       "CallManualOperationLines_ServoPos64Commands"(ManualOperationControl := "ManualOperationControl_U1Em5".axis64Pos[7].commands,
                                                     HmiInterface => "Unit1.Em5.HmiInterface".cmCathodeMainPnP2AxisX.commands);

       "CallManualOperationLines_ServoPos64Commands"(ManualOperationControl := "ManualOperationControl_U1Em5".axis64Pos[8].commands,
                                                     HmiInterface => "Unit1.Em5.HmiInterface".cmCathodeMainPnP1AxisY.commands);

       "CallManualOperationLines_ServoPos64Commands"(ManualOperationControl := "ManualOperationControl_U1Em5".axis64Pos[9].commands,
                                                     HmiInterface => "Unit1.Em5.HmiInterface".cmCathodeMainPnP1AxisZ.commands);

       "CallManualOperationLines_ServoPos64Commands"(ManualOperationControl := "ManualOperationControl_U1Em5".axis64Pos[10].commands,
                                                     HmiInterface => "Unit1.Em5.HmiInterface".cmCathodeMainPnP2AxisZ.commands);

       "CallManualOperationLines_ServoPos64Commands"(ManualOperationControl := "ManualOperationControl_U1Em5".axis64Pos[11].commands,
                                                     HmiInterface => "Unit1.Em5.HmiInterface".cmCathodeAlignTableAxisX.commands);

       "CallManualOperationLines_ServoPos64Commands"(ManualOperationControl := "ManualOperationControl_U1Em5".axis64Pos[12].commands,
                                                     HmiInterface => "Unit1.Em5.HmiInterface".cmCathodeAlignTableAxisY1.commands);

       "CallManualOperationLines_ServoPos64Commands"(ManualOperationControl := "ManualOperationControl_U1Em5".axis64Pos[13].commands,
                                                     HmiInterface => "Unit1.Em5.HmiInterface".cmCathodeAlignTableAxisY2.commands);

       // TwoWayActuator
       "Unit1.Em5.HmiInterface".cmCathodeMainPnP1RotaryCwCcw.commands := "ManualOperationControl_U1Em5".twoWayActuator[1].commands;
       "Unit1.Em5.HmiInterface".cmCathodeMainPnP1SuctionPlateVacuum.commands := "ManualOperationControl_U1Em5".twoWayActuator[2].commands;
       "Unit1.Em5.HmiInterface".cmCathodeMainPnP2SuctionPlateVacuum.commands := "ManualOperationControl_U1Em5".twoWayActuator[3].commands;
       "Unit1.Em5.HmiInterface".cmCathodeAlignTableSuctionPlateVacuum.commands := "ManualOperationControl_U1Em5".twoWayActuator[4].commands;
       "Unit1.Em5.HmiInterface".cmCathodeGlassCleaning.commands := "ManualOperationControl_U1Em5".twoWayActuator[5].commands;
       "Unit1.Em5.HmiInterface".cmCathodeNgPnpUpDown.commands := "ManualOperationControl_U1Em5".twoWayActuator[6].commands;
       "Unit1.Em5.HmiInterface".cmCathodeNgPnp1stFwdBwd.commands := "ManualOperationControl_U1Em5".twoWayActuator[7].commands;
       "Unit1.Em5.HmiInterface".cmCathodeNgPnp2ndFwdBwd.commands := "ManualOperationControl_U1Em5".twoWayActuator[8].commands;
       "Unit1.Em5.HmiInterface".cmCathodeMaintenanceMovingFixFrontRearFwdBwd.commands := "ManualOperationControl_U1Em5".twoWayActuator[9].commands;
       "Unit1.Em5.HmiInterface".cmCathodeNgBoxLiftUpDown.commands := "ManualOperationControl_U1Em5".twoWayActuator[10].commands;
       "Unit1.Em5.HmiInterface".cmCathodeNgBoxLockUpDown.commands := "ManualOperationControl_U1Em5".twoWayActuator[11].commands;
       "Unit1.Em5.HmiInterface".cmCathodeNgPnpVaccum.commands := "ManualOperationControl_U1Em5".twoWayActuator[12].commands;
       "Unit1.Em5.HmiInterface".cmCathodeConveyorCoverFwdBwd.commands := "ManualOperationControl_U1Em5".twoWayActuator[13].commands;

   END_REGION
END_REGION

REGION Network 13: Equipment Module 5
   RUNG wire#powerrail
      "CallManualOperationLines_EM"(disableUnit := #disableUnit1, manualOperationEm := "ManualOperationControl_U1Em5".manualOperationEm, manualOperationEmArea := "ManualOperationControl_U1Em5".manualOperationEmArea, manualOperationCms := "ManualOperationControl_U1Em5".manualOperationCms, Axis := "ManualOperationControl_U1Em5".axis, Axis64Pos := "ManualOperationControl_U1Em5".axis64Pos, AxisSfotCam := "ManualOperationControl_U1Em5".softCam, twoWayAcutor := "ManualOperationControl_U1Em5".twoWayActuator, Status := #StatusEm[5].Status, errorID := #errorIDEm[5].errorID)
   END_RUNG
   // the same network as SCL:
   "CallManualOperationLines_EM"(disableUnit := #disableUnit1,
                           manualOperationEm := "ManualOperationControl_U1Em5".manualOperationEm,
                           manualOperationEmArea := "ManualOperationControl_U1Em5".manualOperationEmArea,
                           manualOperationCms := "ManualOperationControl_U1Em5".manualOperationCms,
                           Axis := "ManualOperationControl_U1Em5".axis,
                           Axis64Pos := "ManualOperationControl_U1Em5".axis64Pos,
                           AxisSfotCam := "ManualOperationControl_U1Em5".softCam,
                           twoWayAcutor := "ManualOperationControl_U1Em5".twoWayActuator,
                           Status := #StatusEm[5].Status,
                           errorID := #errorIDEm[5].errorID);
END_REGION

REGION Network 14 (SCL): Equipment Module 6 Cms Mapping
   REGION Input Mapping
       // Axis
       "ManualOperationControl_U1Em6".axis64Pos[6].monitoring := "Unit1.Em6.HmiInterface".cmFinalRollerFrontAxisX.monitoring;
       "ManualOperationControl_U1Em6".axis64Pos[7].monitoring := "Unit1.Em6.HmiInterface".cmFinalRollerRearAxisX.monitoring;
       "ManualOperationControl_U1Em6".axis64Pos[8].monitoring := "Unit1.Em6.HmiInterface".cmMendrelCathodeFrontAxisY.monitoring;
       "ManualOperationControl_U1Em6".axis64Pos[9].monitoring := "Unit1.Em6.HmiInterface".cmMendrelCathodeFrontAxisZ.monitoring;
       "ManualOperationControl_U1Em6".axis64Pos[10].monitoring := "Unit1.Em6.HmiInterface".cmMendrelAnodeFrontAxisY.monitoring;
       "ManualOperationControl_U1Em6".axis64Pos[11].monitoring := "Unit1.Em6.HmiInterface".cmMendrelAnodeFrontAxisZ.monitoring;
       "ManualOperationControl_U1Em6".axis64Pos[12].monitoring := "Unit1.Em6.HmiInterface".cmMendrelCathodeRearAxisY.monitoring;
       "ManualOperationControl_U1Em6".axis64Pos[13].monitoring := "Unit1.Em6.HmiInterface".cmMendrelCathodeRearAxisZ.monitoring;
       "ManualOperationControl_U1Em6".axis64Pos[14].monitoring := "Unit1.Em6.HmiInterface".cmMendrelAnodeRearAxisY.monitoring;
       "ManualOperationControl_U1Em6".axis64Pos[15].monitoring := "Unit1.Em6.HmiInterface".cmMendrelAnodeRearAxisZ.monitoring;
       "ManualOperationControl_U1Em6".axis64Pos[16].monitoring := "Unit1.Em6.HmiInterface".cmStackTableAxisZ.monitoring;
       "ManualOperationControl_U1Em6".axis64Pos[17].monitoring := "Unit1.Em6.HmiInterface".cmStackTableOutFrontAxisZ.monitoring;
       "ManualOperationControl_U1Em6".axis64Pos[18].monitoring := "Unit1.Em6.HmiInterface".cmStackTableOutRearAxisZ.monitoring;

       "ManualOperationControl_U1Em6".axis64Pos[6].configuration := "Unit1.Em6.HmiInterface".cmFinalRollerFrontAxisX.configuration;
       "ManualOperationControl_U1Em6".axis64Pos[7].configuration := "Unit1.Em6.HmiInterface".cmFinalRollerRearAxisX.configuration;
       "ManualOperationControl_U1Em6".axis64Pos[8].configuration := "Unit1.Em6.HmiInterface".cmMendrelCathodeFrontAxisY.configuration;
       "ManualOperationControl_U1Em6".axis64Pos[9].configuration := "Unit1.Em6.HmiInterface".cmMendrelCathodeFrontAxisZ.configuration;
       "ManualOperationControl_U1Em6".axis64Pos[10].configuration := "Unit1.Em6.HmiInterface".cmMendrelAnodeFrontAxisY.configuration;
       "ManualOperationControl_U1Em6".axis64Pos[11].configuration := "Unit1.Em6.HmiInterface".cmMendrelAnodeFrontAxisZ.configuration;
       "ManualOperationControl_U1Em6".axis64Pos[12].configuration := "Unit1.Em6.HmiInterface".cmMendrelCathodeRearAxisY.configuration;
       "ManualOperationControl_U1Em6".axis64Pos[13].configuration := "Unit1.Em6.HmiInterface".cmMendrelCathodeRearAxisZ.configuration;
       "ManualOperationControl_U1Em6".axis64Pos[14].configuration := "Unit1.Em6.HmiInterface".cmMendrelAnodeRearAxisY.configuration;
       "ManualOperationControl_U1Em6".axis64Pos[15].configuration := "Unit1.Em6.HmiInterface".cmMendrelAnodeRearAxisZ.configuration;
       "ManualOperationControl_U1Em6".axis64Pos[16].configuration := "Unit1.Em6.HmiInterface".cmStackTableAxisZ.configuration;
       "ManualOperationControl_U1Em6".axis64Pos[17].configuration := "Unit1.Em6.HmiInterface".cmStackTableOutFrontAxisZ.configuration;
       "ManualOperationControl_U1Em6".axis64Pos[18].configuration := "Unit1.Em6.HmiInterface".cmStackTableOutRearAxisZ.configuration;

       // SoftCam
       "ManualOperationControl_U1Em6".softCam[6] := "Unit1.Em6.HmiInterface".cm.softCam.finalRollerFrontAxisX;
       "ManualOperationControl_U1Em6".softCam[7] := "Unit1.Em6.HmiInterface".cm.softCam.finalRollerRearAxisX;
       "ManualOperationControl_U1Em6".softCam[8] := "Unit1.Em6.HmiInterface".cm.softCam.mendrelAnodeFrontAxisY;
       "ManualOperationControl_U1Em6".softCam[9] := "Unit1.Em6.HmiInterface".cm.softCam.mendrelAnodeFrontAxisZ;
       "ManualOperationControl_U1Em6".softCam[10] := "Unit1.Em6.HmiInterface".cm.softCam.mendrelAnodeRearAxisY;
       "ManualOperationControl_U1Em6".softCam[11] := "Unit1.Em6.HmiInterface".cm.softCam.mendrelAnodeRearAxisZ;
       "ManualOperationControl_U1Em6".softCam[12] := "Unit1.Em6.HmiInterface".cm.softCam.mendrelCathodeFrontAxisY;
       "ManualOperationControl_U1Em6".softCam[13] := "Unit1.Em6.HmiInterface".cm.softCam.mendrelCathodeFrontAxisZ;
       "ManualOperationControl_U1Em6".softCam[14] := "Unit1.Em6.HmiInterface".cm.softCam.mendrelCathodeRearAxisY;
       "ManualOperationControl_U1Em6".softCam[15] := "Unit1.Em6.HmiInterface".cm.softCam.mendrelCathodeRearAxisZ;
       "ManualOperationControl_U1Em6".softCam[16] := "Unit1.Em6.HmiInterface".cm.softCam.stackTableAxisZ;
       "ManualOperationControl_U1Em6".softCam[17] := "Unit1.Em6.HmiInterface".cm.softCam.stackTableOutFrontAxisZ;
       "ManualOperationControl_U1Em6".softCam[18] := "Unit1.Em6.HmiInterface".cm.softCam.stackTableOutRearAxisZ;

       // TwoWayActuator
       "ManualOperationControl_U1Em6".twoWayActuator[1].monitoring := "Unit1.Em6.HmiInterface".cmMendrelCathodeFrontClamp.monitoring;
       "ManualOperationControl_U1Em6".twoWayActuator[2].monitoring := "Unit1.Em6.HmiInterface".cmMendrelAnodeFrontClamp.monitoring;
       "ManualOperationControl_U1Em6".twoWayActuator[3].monitoring := "Unit1.Em6.HmiInterface".cmMendrelCathodeRearClamp.monitoring;
       "ManualOperationControl_U1Em6".twoWayActuator[4].monitoring := "Unit1.Em6.HmiInterface".cmMendrelAnodeRearClamp.monitoring;
       "ManualOperationControl_U1Em6".twoWayActuator[5].monitoring := "Unit1.Em6.HmiInterface".cmStackTableVaccum.monitoring;
       "ManualOperationControl_U1Em6".twoWayActuator[6].monitoring := "Unit1.Em6.HmiInterface".cmStackTableGapPadUpDown.monitoring;

   END_REGION


   REGION Output Mapping
       // Axis
       "CallManualOperationLines_ServoPos64Commands"(ManualOperationControl := "ManualOperationControl_U1Em6".axis64Pos[6].commands,
                                                     HmiInterface => "Unit1.Em6.HmiInterface".cmFinalRollerFrontAxisX.commands);

       "CallManualOperationLines_ServoPos64Commands"(ManualOperationControl := "ManualOperationControl_U1Em6".axis64Pos[7].commands,
                                                     HmiInterface => "Unit1.Em6.HmiInterface".cmFinalRollerRearAxisX.commands);

       "CallManualOperationLines_ServoPos64Commands"(ManualOperationControl := "ManualOperationControl_U1Em6".axis64Pos[8].commands,
                                                     HmiInterface => "Unit1.Em6.HmiInterface".cmMendrelCathodeFrontAxisY.commands);

       "CallManualOperationLines_ServoPos64Commands"(ManualOperationControl := "ManualOperationControl_U1Em6".axis64Pos[9].commands,
                                                     HmiInterface => "Unit1.Em6.HmiInterface".cmMendrelCathodeFrontAxisZ.commands);

       "CallManualOperationLines_ServoPos64Commands"(ManualOperationControl := "ManualOperationControl_U1Em6".axis64Pos[10].commands,
                                                     HmiInterface => "Unit1.Em6.HmiInterface".cmMendrelAnodeFrontAxisY.commands);

       "CallManualOperationLines_ServoPos64Commands"(ManualOperationControl := "ManualOperationControl_U1Em6".axis64Pos[11].commands,
                                                     HmiInterface => "Unit1.Em6.HmiInterface".cmMendrelAnodeFrontAxisZ.commands);

       "CallManualOperationLines_ServoPos64Commands"(ManualOperationControl := "ManualOperationControl_U1Em6".axis64Pos[12].commands,
                                                     HmiInterface => "Unit1.Em6.HmiInterface".cmMendrelCathodeRearAxisY.commands);

       "CallManualOperationLines_ServoPos64Commands"(ManualOperationControl := "ManualOperationControl_U1Em6".axis64Pos[13].commands,
                                                     HmiInterface => "Unit1.Em6.HmiInterface".cmMendrelCathodeRearAxisZ.commands);

       "CallManualOperationLines_ServoPos64Commands"(ManualOperationControl := "ManualOperationControl_U1Em6".axis64Pos[14].commands,
                                                     HmiInterface => "Unit1.Em6.HmiInterface".cmMendrelAnodeRearAxisY.commands);

       "CallManualOperationLines_ServoPos64Commands"(ManualOperationControl := "ManualOperationControl_U1Em6".axis64Pos[15].commands,
                                                     HmiInterface => "Unit1.Em6.HmiInterface".cmMendrelAnodeRearAxisZ.commands);

       "CallManualOperationLines_ServoPos64Commands"(ManualOperationControl := "ManualOperationControl_U1Em6".axis64Pos[16].commands,
                                                     HmiInterface => "Unit1.Em6.HmiInterface".cmStackTableAxisZ.commands);

       "CallManualOperationLines_ServoPos64Commands"(ManualOperationControl := "ManualOperationControl_U1Em6".axis64Pos[17].commands,
                                                     HmiInterface => "Unit1.Em6.HmiInterface".cmStackTableOutFrontAxisZ.commands);

       "CallManualOperationLines_ServoPos64Commands"(ManualOperationControl := "ManualOperationControl_U1Em6".axis64Pos[18].commands,
                                                     HmiInterface => "Unit1.Em6.HmiInterface".cmStackTableOutRearAxisZ.commands);

       // TwoWayActuator
       "Unit1.Em6.HmiInterface".cmMendrelCathodeFrontClamp.commands := "ManualOperationControl_U1Em6".twoWayActuator[1].commands;
       "Unit1.Em6.HmiInterface".cmMendrelAnodeFrontClamp.commands := "ManualOperationControl_U1Em6".twoWayActuator[2].commands;
       "Unit1.Em6.HmiInterface".cmMendrelCathodeRearClamp.commands := "ManualOperationControl_U1Em6".twoWayActuator[3].commands;
       "Unit1.Em6.HmiInterface".cmMendrelAnodeRearClamp.commands := "ManualOperationControl_U1Em6".twoWayActuator[4].commands;
       "Unit1.Em6.HmiInterface".cmStackTableVaccum.commands := "ManualOperationControl_U1Em6".twoWayActuator[5].commands;
       "Unit1.Em6.HmiInterface".cmStackTableGapPadUpDown.commands := "ManualOperationControl_U1Em6".twoWayActuator[6].commands;
   END_REGION
END_REGION

REGION Network 15: Equipment Module 6
   RUNG wire#powerrail
      "CallManualOperationLines_EM"(disableUnit := #disableUnit1, manualOperationEm := "ManualOperationControl_U1Em6".manualOperationEm, manualOperationEmArea := "ManualOperationControl_U1Em6".manualOperationEmArea, manualOperationCms := "ManualOperationControl_U1Em6".manualOperationCms, Axis := "ManualOperationControl_U1Em6".axis, Axis64Pos := "ManualOperationControl_U1Em6".axis64Pos, AxisSfotCam := "ManualOperationControl_U1Em6".softCam, twoWayAcutor := "ManualOperationControl_U1Em6".twoWayActuator, Status := #StatusEm[6].Status, errorID := #errorIDEm[6].errorID)
   END_RUNG
   // the same network as SCL:
   "CallManualOperationLines_EM"(disableUnit := #disableUnit1,
                           manualOperationEm := "ManualOperationControl_U1Em6".manualOperationEm,
                           manualOperationEmArea := "ManualOperationControl_U1Em6".manualOperationEmArea,
                           manualOperationCms := "ManualOperationControl_U1Em6".manualOperationCms,
                           Axis := "ManualOperationControl_U1Em6".axis,
                           Axis64Pos := "ManualOperationControl_U1Em6".axis64Pos,
                           AxisSfotCam := "ManualOperationControl_U1Em6".softCam,
                           twoWayAcutor := "ManualOperationControl_U1Em6".twoWayActuator,
                           Status := #StatusEm[6].Status,
                           errorID := #errorIDEm[6].errorID);
END_REGION

REGION Network 16 (SCL): Equipment Module 7 Cms Mapping
   REGION Input Mapping
       // Axis
       "ManualOperationControl_U1Em7".axis64Pos[6].monitoring := "Unit1.Em7.HmiInterface".cmSepaClampnCutterAxisX.monitoring;
       "ManualOperationControl_U1Em7".axis64Pos[7].monitoring := "Unit1.Em7.HmiInterface".cmSepaClampnCutterAxisZ.monitoring;
       "ManualOperationControl_U1Em7".axis64Pos[8].monitoring := "Unit1.Em7.HmiInterface".cmSepaGripperAxisX.monitoring;
       "ManualOperationControl_U1Em7".axis64Pos[9].monitoring := "Unit1.Em7.HmiInterface".cmSepaGripperAxisZ.monitoring;
       "ManualOperationControl_U1Em7".axis64Pos[10].monitoring := "Unit1.Em7.HmiInterface".cmSepaGripperAxisC.monitoring;
       "ManualOperationControl_U1Em7".axis64Pos[11].monitoring := "Unit1.Em7.HmiInterface".cmJRWinderFrontAxisY.monitoring;
       "ManualOperationControl_U1Em7".axis64Pos[12].monitoring := "Unit1.Em7.HmiInterface".cmJRWinderRearAxisY.monitoring;
       "ManualOperationControl_U1Em7".axis64Pos[13].monitoring := "Unit1.Em7.HmiInterface".cmJRWinderAxisB.monitoring;
       "ManualOperationControl_U1Em7".axis64Pos[14].monitoring := "Unit1.Em7.HmiInterface".cmJRPusherAxisZ.monitoring;

       "ManualOperationControl_U1Em7".axis64Pos[6].configuration := "Unit1.Em7.HmiInterface".cmSepaClampnCutterAxisX.configuration;
       "ManualOperationControl_U1Em7".axis64Pos[7].configuration := "Unit1.Em7.HmiInterface".cmSepaClampnCutterAxisZ.configuration;
       "ManualOperationControl_U1Em7".axis64Pos[8].configuration := "Unit1.Em7.HmiInterface".cmSepaGripperAxisX.configuration;
       "ManualOperationControl_U1Em7".axis64Pos[9].configuration := "Unit1.Em7.HmiInterface".cmSepaGripperAxisZ.configuration;
       "ManualOperationControl_U1Em7".axis64Pos[10].configuration := "Unit1.Em7.HmiInterface".cmSepaGripperAxisC.configuration;
       "ManualOperationControl_U1Em7".axis64Pos[11].configuration := "Unit1.Em7.HmiInterface".cmJRWinderFrontAxisY.configuration;
       "ManualOperationControl_U1Em7".axis64Pos[12].configuration := "Unit1.Em7.HmiInterface".cmJRWinderRearAxisY.configuration;
       "ManualOperationControl_U1Em7".axis64Pos[13].configuration := "Unit1.Em7.HmiInterface".cmJRWinderAxisB.configuration;
       "ManualOperationControl_U1Em7".axis64Pos[14].configuration := "Unit1.Em7.HmiInterface".cmJRPusherAxisZ.configuration;

       // SoftCam
       "ManualOperationControl_U1Em7".softCam[6] := "Unit1.Em7.HmiInterface".cm.softCam.sepaClampnCutterAxisX;
       "ManualOperationControl_U1Em7".softCam[7] := "Unit1.Em7.HmiInterface".cm.softCam.sepaClampnCutterAxisZ;
       "ManualOperationControl_U1Em7".softCam[8] := "Unit1.Em7.HmiInterface".cm.softCam.sepaGripperAxisX;
       "ManualOperationControl_U1Em7".softCam[9] := "Unit1.Em7.HmiInterface".cm.softCam.sepaGripperAxisZ;
       "ManualOperationControl_U1Em7".softCam[10] := "Unit1.Em7.HmiInterface".cm.softCam.sepaGripperAxisC;
       "ManualOperationControl_U1Em7".softCam[11] := "Unit1.Em7.HmiInterface".cm.softCam.jrWinderRearAxisY;
       "ManualOperationControl_U1Em7".softCam[12] := "Unit1.Em7.HmiInterface".cm.softCam.jrWinderFrontAxisY;
       "ManualOperationControl_U1Em7".softCam[13] := "Unit1.Em7.HmiInterface".cm.softCam.jrWinderAxisB;
       "ManualOperationControl_U1Em7".softCam[14] := "Unit1.Em7.HmiInterface".cm.softCam.jrPusherAxisZ;

       // TwoWayActuator
       "ManualOperationControl_U1Em7".twoWayActuator[1].monitoring := "Unit1.Em7.HmiInterface".cmSepaCutterUpDown.monitoring;
       "ManualOperationControl_U1Em7".twoWayActuator[2].monitoring := "Unit1.Em7.HmiInterface".cmSepaClampTopUpDown.monitoring;
       "ManualOperationControl_U1Em7".twoWayActuator[3].monitoring := "Unit1.Em7.HmiInterface".cmSepaClampBottomUpDown.monitoring;
       "ManualOperationControl_U1Em7".twoWayActuator[4].monitoring := "Unit1.Em7.HmiInterface".cmStackGripperOpenClose.monitoring;
       "ManualOperationControl_U1Em7".twoWayActuator[5].monitoring := "Unit1.Em7.HmiInterface".cmStackGripperFwdBwd.monitoring;
       "ManualOperationControl_U1Em7".twoWayActuator[6].monitoring := "Unit1.Em7.HmiInterface".cmJRWinderClampTopRearUpDown.monitoring;
       "ManualOperationControl_U1Em7".twoWayActuator[7].monitoring := "Unit1.Em7.HmiInterface".cmJRWinderClampBtmRearUpDown.monitoring;
       "ManualOperationControl_U1Em7".twoWayActuator[8].monitoring := "Unit1.Em7.HmiInterface".cmJRWinderClampTopFrontUpDown.monitoring;
       "ManualOperationControl_U1Em7".twoWayActuator[9].monitoring := "Unit1.Em7.HmiInterface".cmJRWinderClampBtmFrontUpDown.monitoring;
       "ManualOperationControl_U1Em7".twoWayActuator[10].monitoring := "Unit1.Em7.HmiInterface".cmPusherRollerFwdBwd.monitoring;

   END_REGION


   REGION Output Mapping
       // Axis
       "CallManualOperationLines_ServoPos64Commands"(ManualOperationControl := "ManualOperationControl_U1Em7".axis64Pos[6].commands,
                                                     HmiInterface => "Unit1.Em7.HmiInterface".cmSepaClampnCutterAxisX.commands);

       "CallManualOperationLines_ServoPos64Commands"(ManualOperationControl := "ManualOperationControl_U1Em7".axis64Pos[7].commands,
                                                     HmiInterface => "Unit1.Em7.HmiInterface".cmSepaClampnCutterAxisZ.commands);

       "CallManualOperationLines_ServoPos64Commands"(ManualOperationControl := "ManualOperationControl_U1Em7".axis64Pos[8].commands,
                                                     HmiInterface => "Unit1.Em7.HmiInterface".cmSepaGripperAxisX.commands);

       "CallManualOperationLines_ServoPos64Commands"(ManualOperationControl := "ManualOperationControl_U1Em7".axis64Pos[9].commands,
                                                     HmiInterface => "Unit1.Em7.HmiInterface".cmSepaGripperAxisZ.commands);

       "CallManualOperationLines_ServoPos64Commands"(ManualOperationControl := "ManualOperationControl_U1Em7".axis64Pos[10].commands,
                                                     HmiInterface => "Unit1.Em7.HmiInterface".cmSepaGripperAxisC.commands);

       "CallManualOperationLines_ServoPos64Commands"(ManualOperationControl := "ManualOperationControl_U1Em7".axis64Pos[11].commands,
                                                     HmiInterface => "Unit1.Em7.HmiInterface".cmJRWinderFrontAxisY.commands);

       "CallManualOperationLines_ServoPos64Commands"(ManualOperationControl := "ManualOperationControl_U1Em7".axis64Pos[12].commands,
                                                     HmiInterface => "Unit1.Em7.HmiInterface".cmJRWinderRearAxisY.commands);

       "CallManualOperationLines_ServoPos64Commands"(ManualOperationControl := "ManualOperationControl_U1Em7".axis64Pos[13].commands,
                                                     HmiInterface => "Unit1.Em7.HmiInterface".cmJRWinderAxisB.commands);

       "CallManualOperationLines_ServoPos64Commands"(ManualOperationControl := "ManualOperationControl_U1Em7".axis64Pos[14].commands,
                                                     HmiInterface => "Unit1.Em7.HmiInterface".cmJRPusherAxisZ.commands);

       // TwoWayActuator
       "Unit1.Em7.HmiInterface".cmSepaCutterUpDown.commands := "ManualOperationControl_U1Em7".twoWayActuator[1].commands;
       "Unit1.Em7.HmiInterface".cmSepaClampTopUpDown.commands := "ManualOperationControl_U1Em7".twoWayActuator[2].commands;
       "Unit1.Em7.HmiInterface".cmSepaClampBottomUpDown.commands := "ManualOperationControl_U1Em7".twoWayActuator[3].commands;
       "Unit1.Em7.HmiInterface".cmStackGripperOpenClose.commands := "ManualOperationControl_U1Em7".twoWayActuator[4].commands;
       "Unit1.Em7.HmiInterface".cmStackGripperFwdBwd.commands := "ManualOperationControl_U1Em7".twoWayActuator[5].commands;
       "Unit1.Em7.HmiInterface".cmJRWinderClampTopRearUpDown.commands := "ManualOperationControl_U1Em7".twoWayActuator[6].commands;
       "Unit1.Em7.HmiInterface".cmJRWinderClampBtmRearUpDown.commands := "ManualOperationControl_U1Em7".twoWayActuator[7].commands;
       "Unit1.Em7.HmiInterface".cmJRWinderClampTopFrontUpDown.commands := "ManualOperationControl_U1Em7".twoWayActuator[8].commands;
       "Unit1.Em7.HmiInterface".cmJRWinderClampBtmFrontUpDown.commands := "ManualOperationControl_U1Em7".twoWayActuator[9].commands;
       "Unit1.Em7.HmiInterface".cmPusherRollerFwdBwd.commands := "ManualOperationControl_U1Em7".twoWayActuator[10].commands;

   END_REGION
END_REGION

REGION Network 17: Equipment Module 7
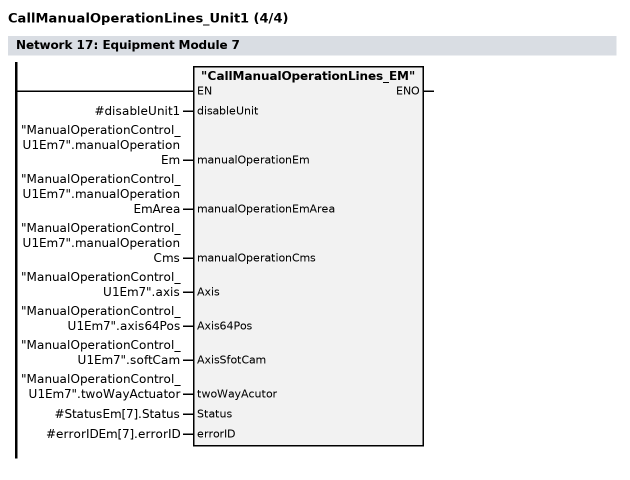
   RUNG wire#powerrail
      "CallManualOperationLines_EM"(disableUnit := #disableUnit1, manualOperationEm := "ManualOperationControl_U1Em7".manualOperationEm, manualOperationEmArea := "ManualOperationControl_U1Em7".manualOperationEmArea, manualOperationCms := "ManualOperationControl_U1Em7".manualOperationCms, Axis := "ManualOperationControl_U1Em7".axis, Axis64Pos := "ManualOperationControl_U1Em7".axis64Pos, AxisSfotCam := "ManualOperationControl_U1Em7".softCam, twoWayAcutor := "ManualOperationControl_U1Em7".twoWayActuator, Status := #StatusEm[7].Status, errorID := #errorIDEm[7].errorID)
   END_RUNG
   // the same network as SCL:
   "CallManualOperationLines_EM"(disableUnit := #disableUnit1,
                           manualOperationEm := "ManualOperationControl_U1Em7".manualOperationEm,
                           manualOperationEmArea := "ManualOperationControl_U1Em7".manualOperationEmArea,
                           manualOperationCms := "ManualOperationControl_U1Em7".manualOperationCms,
                           Axis := "ManualOperationControl_U1Em7".axis,
                           Axis64Pos := "ManualOperationControl_U1Em7".axis64Pos,
                           AxisSfotCam := "ManualOperationControl_U1Em7".softCam,
                           twoWayAcutor := "ManualOperationControl_U1Em7".twoWayActuator,
                           Status := #StatusEm[7].Status,
                           errorID := #errorIDEm[7].errorID);
END_REGION
END_FUNCTION

FUNCTION "CallManualOperationLines_EM" : Void   // FC82, LAD
// stored: SetENOAutomatically false
   VAR_INPUT
      disableUnit : Bool;
   END_VAR
   VAR_IN_OUT
      manualOperationEm : "LAF_typeManEm";
      manualOperationEmArea : Array[*] of "LAF_typeManOperationArea";
      manualOperationCms : Array[*] of "LAF_typeManOperation";
      Axis : Array[*] of "LBC_typeAxisControlInterface";
      Axis64Pos : Array[*] of "LBC_typeAxis64PosInterface";
      AxisSfotCam : Array[*] of "LER_typeSoftCamInterface2";
      twoWayAcutor : Array[*] of "LBC_typeTwoWayActuatorInterface";
      Status : Array[*] of Word;
      errorID : Array[*] of Word;
   END_VAR
   VAR_TEMP
      tempLowerBoundAxis : Int;
      tempUpperBoundAxis : Int;
      tempLowerBoundAxis64Pos : Int;
      tempUpperBoundAxis64Pos : Int;
      tempLowerBoundTwoWayAct : Int;
      tempUpperBoundTwoWayAct : Int;
      tempEnd : Bool;
   END_VAR
BEGIN

REGION Network 1: Detect lower and upper bound of the array for further processing
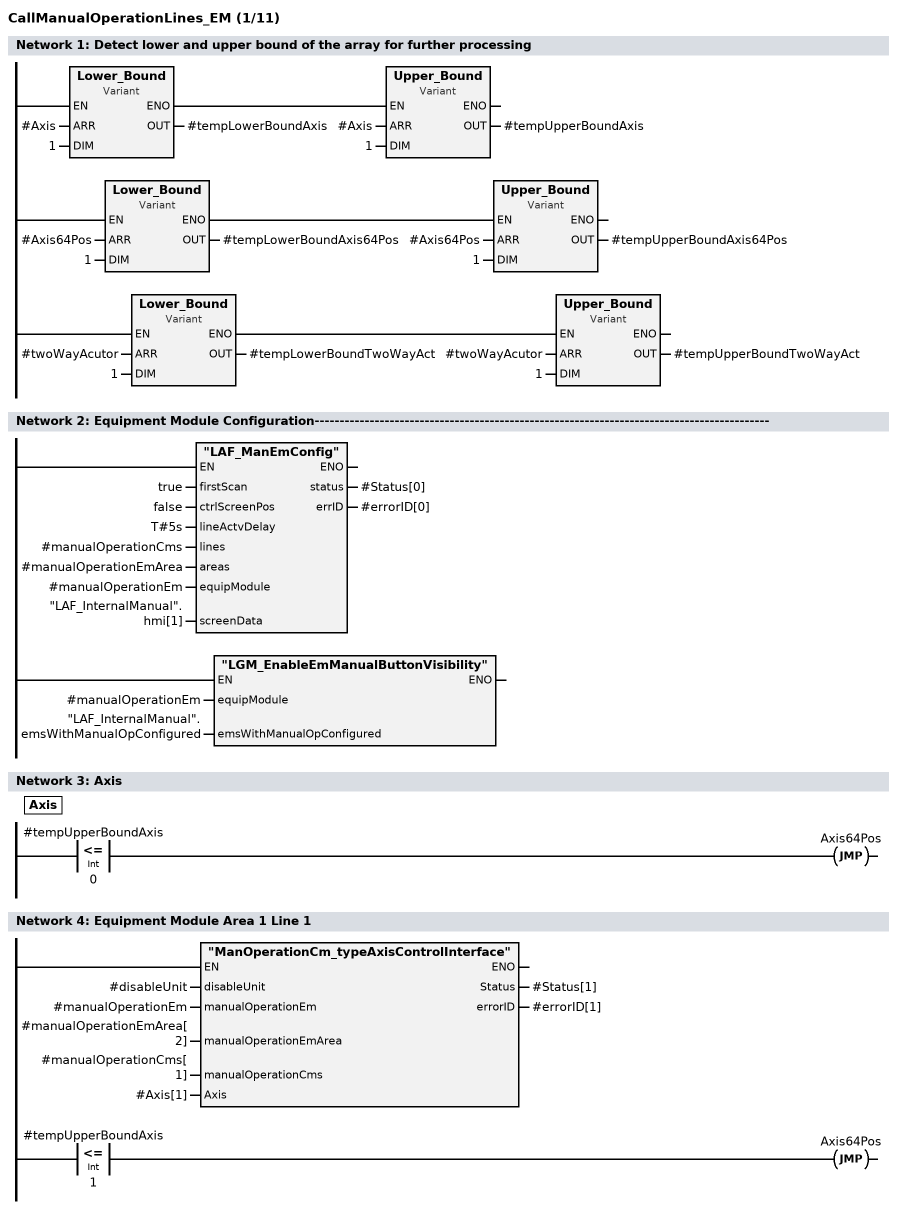
   // no SCL statement known for Lower_Bound, Upper_Bound: written as a call
   // ENO of a box is taken as its EN; it also drops when the box reports an error
   Lower_Bound(arr := #Axis, dim := 1, out => #tempLowerBoundAxis);
   Upper_Bound(arr := #Axis, dim := 1, out => #tempUpperBoundAxis);
   Lower_Bound(arr := #Axis64Pos, dim := 1, out => #tempLowerBoundAxis64Pos);
   Upper_Bound(arr := #Axis64Pos, dim := 1, out => #tempUpperBoundAxis64Pos);
   Lower_Bound(arr := #twoWayAcutor, dim := 1, out => #tempLowerBoundTwoWayAct);
   Upper_Bound(arr := #twoWayAcutor, dim := 1, out => #tempUpperBoundTwoWayAct);
END_REGION

REGION Network 2: Equipment Module Configuration-------------------------------------------------------------------------------------------
   RUNG wire#powerrail
      "LAF_ManEmConfig"(firstScan := true, ctrlScreenPos := false, lineActvDelay := T#5s, lines := #manualOperationCms, areas := #manualOperationEmArea, equipModule := #manualOperationEm, screenData := "LAF_InternalManual".hmi[1], status => #Status[0], errID => #errorID[0])
   END_RUNG
   RUNG wire#powerrail
      "LGM_EnableEmManualButtonVisibility"(equipModule := #manualOperationEm, emsWithManualOpConfigured := "LAF_InternalManual".emsWithManualOpConfigured)
   END_RUNG
   // the same network as SCL:
   "LAF_ManEmConfig"(firstScan := true,
                     ctrlScreenPos := false,
                     lineActvDelay := T#5s,
                     lines := #manualOperationCms,
                     areas := #manualOperationEmArea,
                     equipModule := #manualOperationEm,
                     screenData := "LAF_InternalManual".hmi[1],
                     status => #Status[0],
                     errID => #errorID[0]);
   "LGM_EnableEmManualButtonVisibility"(equipModule := #manualOperationEm,
                           emsWithManualOpConfigured := "LAF_InternalManual".emsWithManualOpConfigured);
END_REGION

REGION Network 3: Axis
   Label( Axis )
   RUNG wire#powerrail
      { S7_Templates := "SrcType := Int" } LE_Contact(in1 := #tempUpperBoundAxis, in2 := 0)
      JumpCoil( Axis64Pos )
   END_RUNG
   // the same network as SCL:
   Axis:
   IF #tempUpperBoundAxis <= 0 THEN GOTO Axis64Pos; END_IF;
END_REGION

REGION Network 4: Equipment Module Area 1 Line 1
   RUNG wire#powerrail
      "ManOperationCm_typeAxisControlInterface"(disableUnit := #disableUnit, manualOperationEm := #manualOperationEm, manualOperationEmArea := #manualOperationEmArea[2], manualOperationCms := #manualOperationCms[1], Axis := #Axis[1], Status => #Status[1], errorID => #errorID[1])
   END_RUNG
   RUNG wire#powerrail
      { S7_Templates := "SrcType := Int" } LE_Contact(in1 := #tempUpperBoundAxis, in2 := 1)
      JumpCoil( Axis64Pos )
   END_RUNG
   // the same network as SCL:
   "ManOperationCm_typeAxisControlInterface"(disableUnit := #disableUnit,
                           manualOperationEm := #manualOperationEm,
                           manualOperationEmArea := #manualOperationEmArea[2],
                           manualOperationCms := #manualOperationCms[1],
                           Axis := #Axis[1],
                           Status => #Status[1],
                           errorID => #errorID[1]);
   IF #tempUpperBoundAxis <= 1 THEN GOTO Axis64Pos; END_IF;
END_REGION

REGION Network 5: Equipment Module Area 1 Line 2
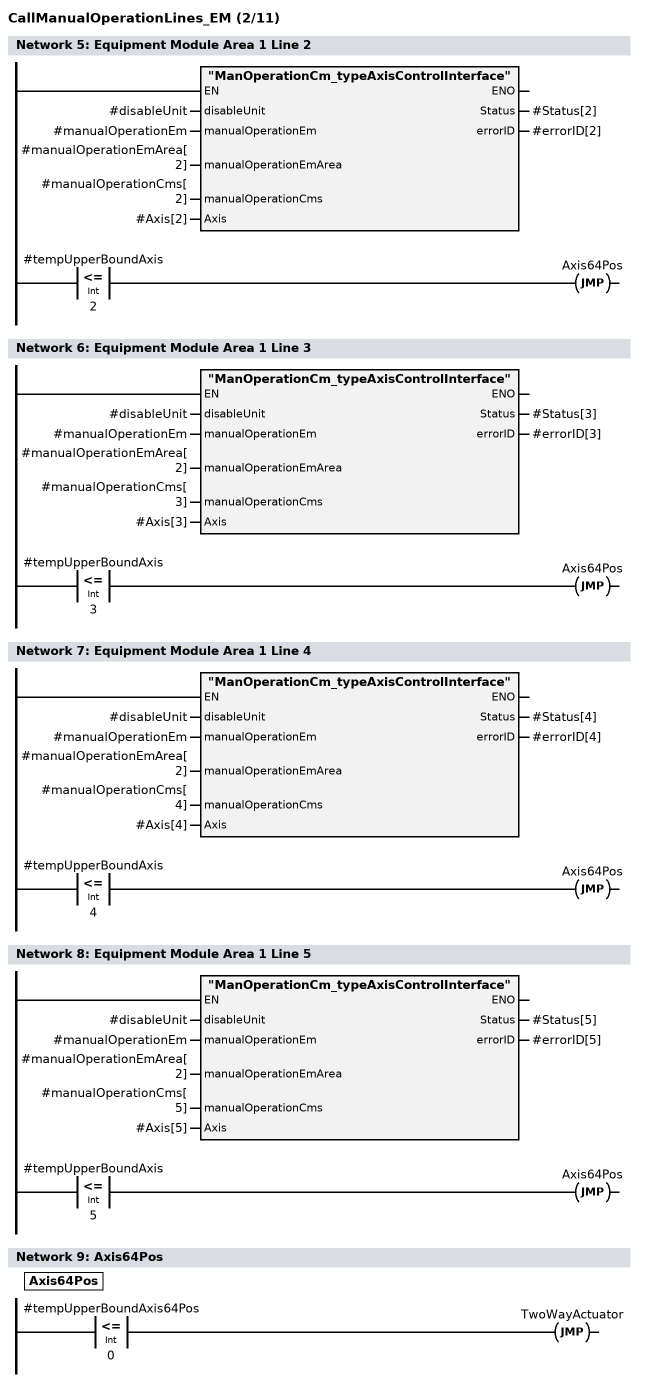
   RUNG wire#powerrail
      "ManOperationCm_typeAxisControlInterface"(disableUnit := #disableUnit, manualOperationEm := #manualOperationEm, manualOperationEmArea := #manualOperationEmArea[2], manualOperationCms := #manualOperationCms[2], Axis := #Axis[2], Status => #Status[2], errorID => #errorID[2])
   END_RUNG
   RUNG wire#powerrail
      { S7_Templates := "SrcType := Int" } LE_Contact(in1 := #tempUpperBoundAxis, in2 := 2)
      JumpCoil( Axis64Pos )
   END_RUNG
   // the same network as SCL:
   "ManOperationCm_typeAxisControlInterface"(disableUnit := #disableUnit,
                           manualOperationEm := #manualOperationEm,
                           manualOperationEmArea := #manualOperationEmArea[2],
                           manualOperationCms := #manualOperationCms[2],
                           Axis := #Axis[2],
                           Status => #Status[2],
                           errorID => #errorID[2]);
   IF #tempUpperBoundAxis <= 2 THEN GOTO Axis64Pos; END_IF;
END_REGION

REGION Network 6: Equipment Module Area 1 Line 3
   RUNG wire#powerrail
      "ManOperationCm_typeAxisControlInterface"(disableUnit := #disableUnit, manualOperationEm := #manualOperationEm, manualOperationEmArea := #manualOperationEmArea[2], manualOperationCms := #manualOperationCms[3], Axis := #Axis[3], Status => #Status[3], errorID => #errorID[3])
   END_RUNG
   RUNG wire#powerrail
      { S7_Templates := "SrcType := Int" } LE_Contact(in1 := #tempUpperBoundAxis, in2 := 3)
      JumpCoil( Axis64Pos )
   END_RUNG
   // the same network as SCL:
   "ManOperationCm_typeAxisControlInterface"(disableUnit := #disableUnit,
                           manualOperationEm := #manualOperationEm,
                           manualOperationEmArea := #manualOperationEmArea[2],
                           manualOperationCms := #manualOperationCms[3],
                           Axis := #Axis[3],
                           Status => #Status[3],
                           errorID => #errorID[3]);
   IF #tempUpperBoundAxis <= 3 THEN GOTO Axis64Pos; END_IF;
END_REGION

REGION Network 7: Equipment Module Area 1 Line 4
   RUNG wire#powerrail
      "ManOperationCm_typeAxisControlInterface"(disableUnit := #disableUnit, manualOperationEm := #manualOperationEm, manualOperationEmArea := #manualOperationEmArea[2], manualOperationCms := #manualOperationCms[4], Axis := #Axis[4], Status => #Status[4], errorID => #errorID[4])
   END_RUNG
   RUNG wire#powerrail
      { S7_Templates := "SrcType := Int" } LE_Contact(in1 := #tempUpperBoundAxis, in2 := 4)
      JumpCoil( Axis64Pos )
   END_RUNG
   // the same network as SCL:
   "ManOperationCm_typeAxisControlInterface"(disableUnit := #disableUnit,
                           manualOperationEm := #manualOperationEm,
                           manualOperationEmArea := #manualOperationEmArea[2],
                           manualOperationCms := #manualOperationCms[4],
                           Axis := #Axis[4],
                           Status => #Status[4],
                           errorID => #errorID[4]);
   IF #tempUpperBoundAxis <= 4 THEN GOTO Axis64Pos; END_IF;
END_REGION

REGION Network 8: Equipment Module Area 1 Line 5
   RUNG wire#powerrail
      "ManOperationCm_typeAxisControlInterface"(disableUnit := #disableUnit, manualOperationEm := #manualOperationEm, manualOperationEmArea := #manualOperationEmArea[2], manualOperationCms := #manualOperationCms[5], Axis := #Axis[5], Status => #Status[5], errorID => #errorID[5])
   END_RUNG
   RUNG wire#powerrail
      { S7_Templates := "SrcType := Int" } LE_Contact(in1 := #tempUpperBoundAxis, in2 := 5)
      JumpCoil( Axis64Pos )
   END_RUNG
   // the same network as SCL:
   "ManOperationCm_typeAxisControlInterface"(disableUnit := #disableUnit,
                           manualOperationEm := #manualOperationEm,
                           manualOperationEmArea := #manualOperationEmArea[2],
                           manualOperationCms := #manualOperationCms[5],
                           Axis := #Axis[5],
                           Status => #Status[5],
                           errorID => #errorID[5]);
   IF #tempUpperBoundAxis <= 5 THEN GOTO Axis64Pos; END_IF;
END_REGION

REGION Network 9: Axis64Pos
   Label( Axis64Pos )
   RUNG wire#powerrail
      { S7_Templates := "SrcType := Int" } LE_Contact(in1 := #tempUpperBoundAxis64Pos, in2 := 0)
      JumpCoil( TwoWayActuator )
   END_RUNG
   // the same network as SCL:
   Axis64Pos:
   IF #tempUpperBoundAxis64Pos <= 0 THEN GOTO TwoWayActuator; END_IF;
END_REGION

REGION Network 10: Equipment Module Area 1 Line 6
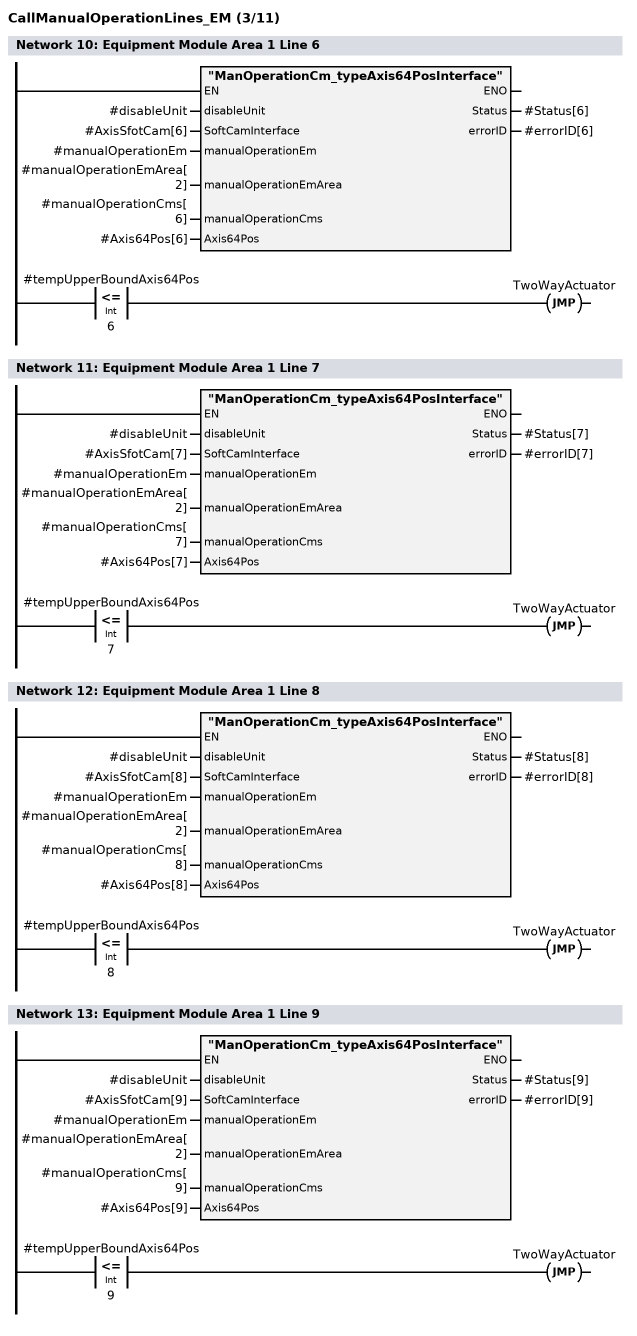
   RUNG wire#powerrail
      "ManOperationCm_typeAxis64PosInterface"(disableUnit := #disableUnit, SoftCamInterface := #AxisSfotCam[6], manualOperationEm := #manualOperationEm, manualOperationEmArea := #manualOperationEmArea[2], manualOperationCms := #manualOperationCms[6], Axis64Pos := #Axis64Pos[6], Status => #Status[6], errorID => #errorID[6])
   END_RUNG
   RUNG wire#powerrail
      { S7_Templates := "SrcType := Int" } LE_Contact(in1 := #tempUpperBoundAxis64Pos, in2 := 6)
      JumpCoil( TwoWayActuator )
   END_RUNG
   // the same network as SCL:
   "ManOperationCm_typeAxis64PosInterface"(disableUnit := #disableUnit,
                           SoftCamInterface := #AxisSfotCam[6],
                           manualOperationEm := #manualOperationEm,
                           manualOperationEmArea := #manualOperationEmArea[2],
                           manualOperationCms := #manualOperationCms[6],
                           Axis64Pos := #Axis64Pos[6],
                           Status => #Status[6],
                           errorID => #errorID[6]);
   IF #tempUpperBoundAxis64Pos <= 6 THEN GOTO TwoWayActuator; END_IF;
END_REGION

REGION Network 11: Equipment Module Area 1 Line 7
   RUNG wire#powerrail
      "ManOperationCm_typeAxis64PosInterface"(disableUnit := #disableUnit, SoftCamInterface := #AxisSfotCam[7], manualOperationEm := #manualOperationEm, manualOperationEmArea := #manualOperationEmArea[2], manualOperationCms := #manualOperationCms[7], Axis64Pos := #Axis64Pos[7], Status => #Status[7], errorID => #errorID[7])
   END_RUNG
   RUNG wire#powerrail
      { S7_Templates := "SrcType := Int" } LE_Contact(in1 := #tempUpperBoundAxis64Pos, in2 := 7)
      JumpCoil( TwoWayActuator )
   END_RUNG
   // the same network as SCL:
   "ManOperationCm_typeAxis64PosInterface"(disableUnit := #disableUnit,
                           SoftCamInterface := #AxisSfotCam[7],
                           manualOperationEm := #manualOperationEm,
                           manualOperationEmArea := #manualOperationEmArea[2],
                           manualOperationCms := #manualOperationCms[7],
                           Axis64Pos := #Axis64Pos[7],
                           Status => #Status[7],
                           errorID => #errorID[7]);
   IF #tempUpperBoundAxis64Pos <= 7 THEN GOTO TwoWayActuator; END_IF;
END_REGION

REGION Network 12: Equipment Module Area 1 Line 8
   RUNG wire#powerrail
      "ManOperationCm_typeAxis64PosInterface"(disableUnit := #disableUnit, SoftCamInterface := #AxisSfotCam[8], manualOperationEm := #manualOperationEm, manualOperationEmArea := #manualOperationEmArea[2], manualOperationCms := #manualOperationCms[8], Axis64Pos := #Axis64Pos[8], Status => #Status[8], errorID => #errorID[8])
   END_RUNG
   RUNG wire#powerrail
      { S7_Templates := "SrcType := Int" } LE_Contact(in1 := #tempUpperBoundAxis64Pos, in2 := 8)
      JumpCoil( TwoWayActuator )
   END_RUNG
   // the same network as SCL:
   "ManOperationCm_typeAxis64PosInterface"(disableUnit := #disableUnit,
                           SoftCamInterface := #AxisSfotCam[8],
                           manualOperationEm := #manualOperationEm,
                           manualOperationEmArea := #manualOperationEmArea[2],
                           manualOperationCms := #manualOperationCms[8],
                           Axis64Pos := #Axis64Pos[8],
                           Status => #Status[8],
                           errorID => #errorID[8]);
   IF #tempUpperBoundAxis64Pos <= 8 THEN GOTO TwoWayActuator; END_IF;
END_REGION

REGION Network 13: Equipment Module Area 1 Line 9
   RUNG wire#powerrail
      "ManOperationCm_typeAxis64PosInterface"(disableUnit := #disableUnit, SoftCamInterface := #AxisSfotCam[9], manualOperationEm := #manualOperationEm, manualOperationEmArea := #manualOperationEmArea[2], manualOperationCms := #manualOperationCms[9], Axis64Pos := #Axis64Pos[9], Status => #Status[9], errorID => #errorID[9])
   END_RUNG
   RUNG wire#powerrail
      { S7_Templates := "SrcType := Int" } LE_Contact(in1 := #tempUpperBoundAxis64Pos, in2 := 9)
      JumpCoil( TwoWayActuator )
   END_RUNG
   // the same network as SCL:
   "ManOperationCm_typeAxis64PosInterface"(disableUnit := #disableUnit,
                           SoftCamInterface := #AxisSfotCam[9],
                           manualOperationEm := #manualOperationEm,
                           manualOperationEmArea := #manualOperationEmArea[2],
                           manualOperationCms := #manualOperationCms[9],
                           Axis64Pos := #Axis64Pos[9],
                           Status => #Status[9],
                           errorID => #errorID[9]);
   IF #tempUpperBoundAxis64Pos <= 9 THEN GOTO TwoWayActuator; END_IF;
END_REGION

REGION Network 14: Equipment Module Area 1 Line 10
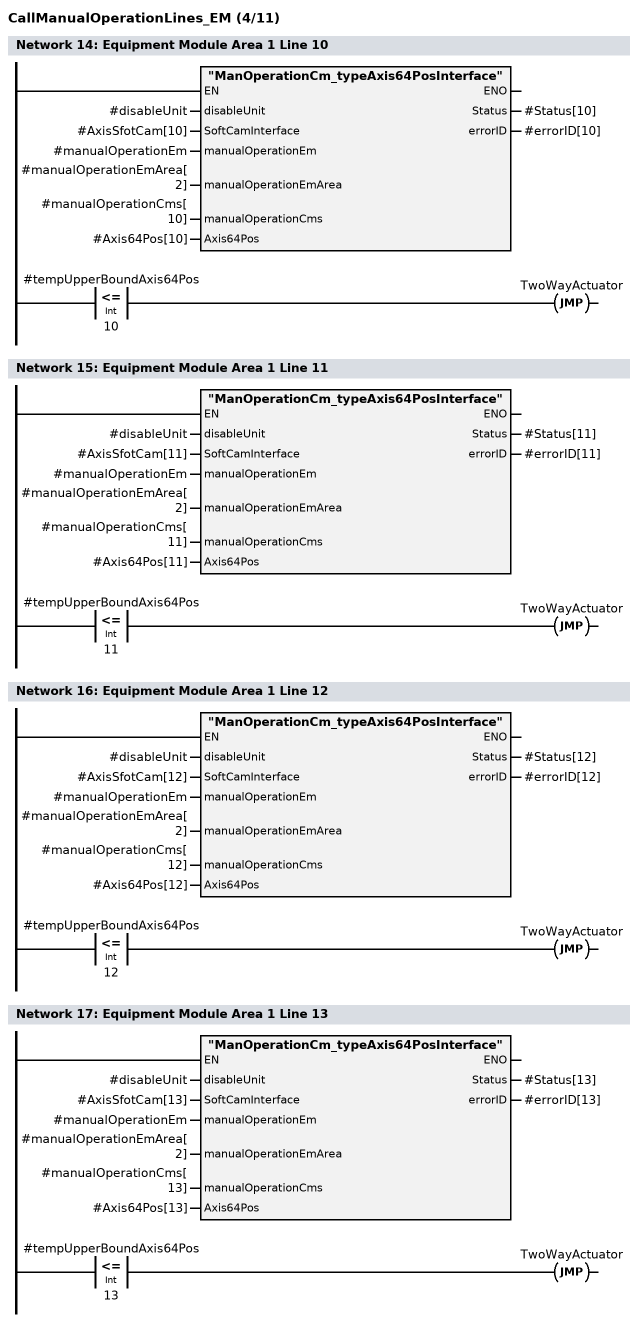
   RUNG wire#powerrail
      "ManOperationCm_typeAxis64PosInterface"(disableUnit := #disableUnit, SoftCamInterface := #AxisSfotCam[10], manualOperationEm := #manualOperationEm, manualOperationEmArea := #manualOperationEmArea[2], manualOperationCms := #manualOperationCms[10], Axis64Pos := #Axis64Pos[10], Status => #Status[10], errorID => #errorID[10])
   END_RUNG
   RUNG wire#powerrail
      { S7_Templates := "SrcType := Int" } LE_Contact(in1 := #tempUpperBoundAxis64Pos, in2 := 10)
      JumpCoil( TwoWayActuator )
   END_RUNG
   // the same network as SCL:
   "ManOperationCm_typeAxis64PosInterface"(disableUnit := #disableUnit,
                           SoftCamInterface := #AxisSfotCam[10],
                           manualOperationEm := #manualOperationEm,
                           manualOperationEmArea := #manualOperationEmArea[2],
                           manualOperationCms := #manualOperationCms[10],
                           Axis64Pos := #Axis64Pos[10],
                           Status => #Status[10],
                           errorID => #errorID[10]);
   IF #tempUpperBoundAxis64Pos <= 10 THEN GOTO TwoWayActuator; END_IF;
END_REGION

REGION Network 15: Equipment Module Area 1 Line 11
   RUNG wire#powerrail
      "ManOperationCm_typeAxis64PosInterface"(disableUnit := #disableUnit, SoftCamInterface := #AxisSfotCam[11], manualOperationEm := #manualOperationEm, manualOperationEmArea := #manualOperationEmArea[2], manualOperationCms := #manualOperationCms[11], Axis64Pos := #Axis64Pos[11], Status => #Status[11], errorID => #errorID[11])
   END_RUNG
   RUNG wire#powerrail
      { S7_Templates := "SrcType := Int" } LE_Contact(in1 := #tempUpperBoundAxis64Pos, in2 := 11)
      JumpCoil( TwoWayActuator )
   END_RUNG
   // the same network as SCL:
   "ManOperationCm_typeAxis64PosInterface"(disableUnit := #disableUnit,
                           SoftCamInterface := #AxisSfotCam[11],
                           manualOperationEm := #manualOperationEm,
                           manualOperationEmArea := #manualOperationEmArea[2],
                           manualOperationCms := #manualOperationCms[11],
                           Axis64Pos := #Axis64Pos[11],
                           Status => #Status[11],
                           errorID => #errorID[11]);
   IF #tempUpperBoundAxis64Pos <= 11 THEN GOTO TwoWayActuator; END_IF;
END_REGION

REGION Network 16: Equipment Module Area 1 Line 12
   RUNG wire#powerrail
      "ManOperationCm_typeAxis64PosInterface"(disableUnit := #disableUnit, SoftCamInterface := #AxisSfotCam[12], manualOperationEm := #manualOperationEm, manualOperationEmArea := #manualOperationEmArea[2], manualOperationCms := #manualOperationCms[12], Axis64Pos := #Axis64Pos[12], Status => #Status[12], errorID => #errorID[12])
   END_RUNG
   RUNG wire#powerrail
      { S7_Templates := "SrcType := Int" } LE_Contact(in1 := #tempUpperBoundAxis64Pos, in2 := 12)
      JumpCoil( TwoWayActuator )
   END_RUNG
   // the same network as SCL:
   "ManOperationCm_typeAxis64PosInterface"(disableUnit := #disableUnit,
                           SoftCamInterface := #AxisSfotCam[12],
                           manualOperationEm := #manualOperationEm,
                           manualOperationEmArea := #manualOperationEmArea[2],
                           manualOperationCms := #manualOperationCms[12],
                           Axis64Pos := #Axis64Pos[12],
                           Status => #Status[12],
                           errorID => #errorID[12]);
   IF #tempUpperBoundAxis64Pos <= 12 THEN GOTO TwoWayActuator; END_IF;
END_REGION

REGION Network 17: Equipment Module Area 1 Line 13
   RUNG wire#powerrail
      "ManOperationCm_typeAxis64PosInterface"(disableUnit := #disableUnit, SoftCamInterface := #AxisSfotCam[13], manualOperationEm := #manualOperationEm, manualOperationEmArea := #manualOperationEmArea[2], manualOperationCms := #manualOperationCms[13], Axis64Pos := #Axis64Pos[13], Status => #Status[13], errorID => #errorID[13])
   END_RUNG
   RUNG wire#powerrail
      { S7_Templates := "SrcType := Int" } LE_Contact(in1 := #tempUpperBoundAxis64Pos, in2 := 13)
      JumpCoil( TwoWayActuator )
   END_RUNG
   // the same network as SCL:
   "ManOperationCm_typeAxis64PosInterface"(disableUnit := #disableUnit,
                           SoftCamInterface := #AxisSfotCam[13],
                           manualOperationEm := #manualOperationEm,
                           manualOperationEmArea := #manualOperationEmArea[2],
                           manualOperationCms := #manualOperationCms[13],
                           Axis64Pos := #Axis64Pos[13],
                           Status => #Status[13],
                           errorID => #errorID[13]);
   IF #tempUpperBoundAxis64Pos <= 13 THEN GOTO TwoWayActuator; END_IF;
END_REGION

REGION Network 18: Equipment Module Area 1 Line 14
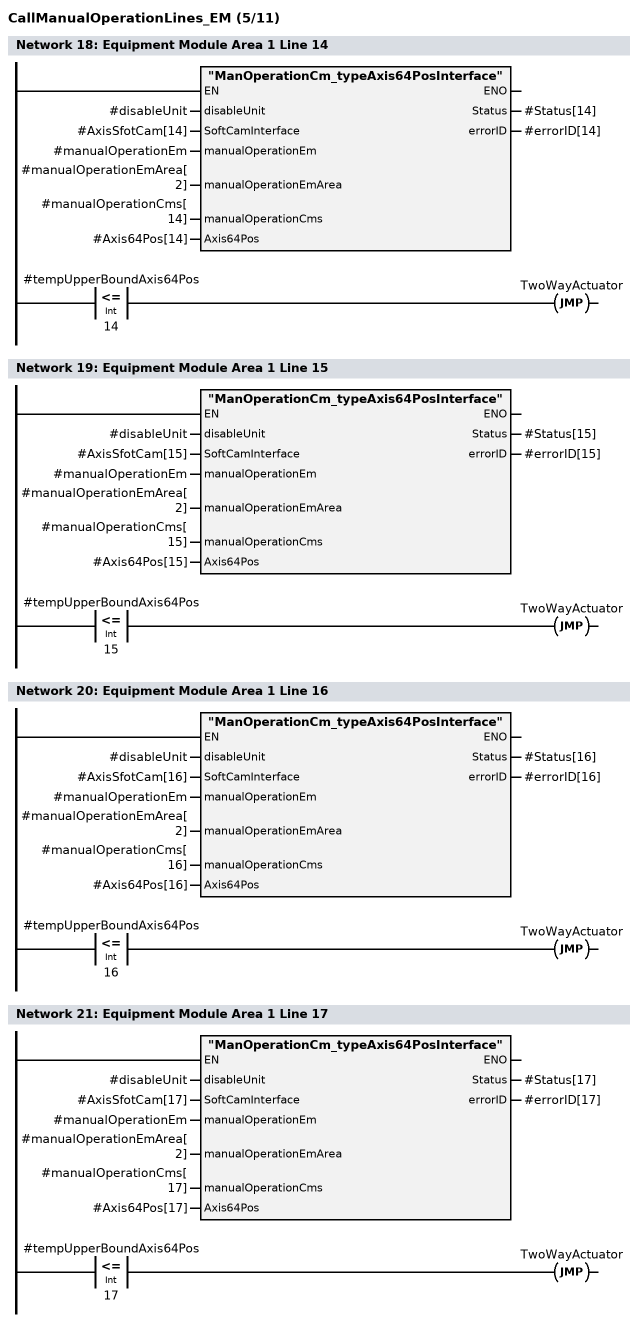
   RUNG wire#powerrail
      "ManOperationCm_typeAxis64PosInterface"(disableUnit := #disableUnit, SoftCamInterface := #AxisSfotCam[14], manualOperationEm := #manualOperationEm, manualOperationEmArea := #manualOperationEmArea[2], manualOperationCms := #manualOperationCms[14], Axis64Pos := #Axis64Pos[14], Status => #Status[14], errorID => #errorID[14])
   END_RUNG
   RUNG wire#powerrail
      { S7_Templates := "SrcType := Int" } LE_Contact(in1 := #tempUpperBoundAxis64Pos, in2 := 14)
      JumpCoil( TwoWayActuator )
   END_RUNG
   // the same network as SCL:
   "ManOperationCm_typeAxis64PosInterface"(disableUnit := #disableUnit,
                           SoftCamInterface := #AxisSfotCam[14],
                           manualOperationEm := #manualOperationEm,
                           manualOperationEmArea := #manualOperationEmArea[2],
                           manualOperationCms := #manualOperationCms[14],
                           Axis64Pos := #Axis64Pos[14],
                           Status => #Status[14],
                           errorID => #errorID[14]);
   IF #tempUpperBoundAxis64Pos <= 14 THEN GOTO TwoWayActuator; END_IF;
END_REGION

REGION Network 19: Equipment Module Area 1 Line 15
   RUNG wire#powerrail
      "ManOperationCm_typeAxis64PosInterface"(disableUnit := #disableUnit, SoftCamInterface := #AxisSfotCam[15], manualOperationEm := #manualOperationEm, manualOperationEmArea := #manualOperationEmArea[2], manualOperationCms := #manualOperationCms[15], Axis64Pos := #Axis64Pos[15], Status => #Status[15], errorID => #errorID[15])
   END_RUNG
   RUNG wire#powerrail
      { S7_Templates := "SrcType := Int" } LE_Contact(in1 := #tempUpperBoundAxis64Pos, in2 := 15)
      JumpCoil( TwoWayActuator )
   END_RUNG
   // the same network as SCL:
   "ManOperationCm_typeAxis64PosInterface"(disableUnit := #disableUnit,
                           SoftCamInterface := #AxisSfotCam[15],
                           manualOperationEm := #manualOperationEm,
                           manualOperationEmArea := #manualOperationEmArea[2],
                           manualOperationCms := #manualOperationCms[15],
                           Axis64Pos := #Axis64Pos[15],
                           Status => #Status[15],
                           errorID => #errorID[15]);
   IF #tempUpperBoundAxis64Pos <= 15 THEN GOTO TwoWayActuator; END_IF;
END_REGION

REGION Network 20: Equipment Module Area 1 Line 16
   RUNG wire#powerrail
      "ManOperationCm_typeAxis64PosInterface"(disableUnit := #disableUnit, SoftCamInterface := #AxisSfotCam[16], manualOperationEm := #manualOperationEm, manualOperationEmArea := #manualOperationEmArea[2], manualOperationCms := #manualOperationCms[16], Axis64Pos := #Axis64Pos[16], Status => #Status[16], errorID => #errorID[16])
   END_RUNG
   RUNG wire#powerrail
      { S7_Templates := "SrcType := Int" } LE_Contact(in1 := #tempUpperBoundAxis64Pos, in2 := 16)
      JumpCoil( TwoWayActuator )
   END_RUNG
   // the same network as SCL:
   "ManOperationCm_typeAxis64PosInterface"(disableUnit := #disableUnit,
                           SoftCamInterface := #AxisSfotCam[16],
                           manualOperationEm := #manualOperationEm,
                           manualOperationEmArea := #manualOperationEmArea[2],
                           manualOperationCms := #manualOperationCms[16],
                           Axis64Pos := #Axis64Pos[16],
                           Status => #Status[16],
                           errorID => #errorID[16]);
   IF #tempUpperBoundAxis64Pos <= 16 THEN GOTO TwoWayActuator; END_IF;
END_REGION

REGION Network 21: Equipment Module Area 1 Line 17
   RUNG wire#powerrail
      "ManOperationCm_typeAxis64PosInterface"(disableUnit := #disableUnit, SoftCamInterface := #AxisSfotCam[17], manualOperationEm := #manualOperationEm, manualOperationEmArea := #manualOperationEmArea[2], manualOperationCms := #manualOperationCms[17], Axis64Pos := #Axis64Pos[17], Status => #Status[17], errorID => #errorID[17])
   END_RUNG
   RUNG wire#powerrail
      { S7_Templates := "SrcType := Int" } LE_Contact(in1 := #tempUpperBoundAxis64Pos, in2 := 17)
      JumpCoil( TwoWayActuator )
   END_RUNG
   // the same network as SCL:
   "ManOperationCm_typeAxis64PosInterface"(disableUnit := #disableUnit,
                           SoftCamInterface := #AxisSfotCam[17],
                           manualOperationEm := #manualOperationEm,
                           manualOperationEmArea := #manualOperationEmArea[2],
                           manualOperationCms := #manualOperationCms[17],
                           Axis64Pos := #Axis64Pos[17],
                           Status => #Status[17],
                           errorID => #errorID[17]);
   IF #tempUpperBoundAxis64Pos <= 17 THEN GOTO TwoWayActuator; END_IF;
END_REGION

REGION Network 22: Equipment Module Area 1 Line 18
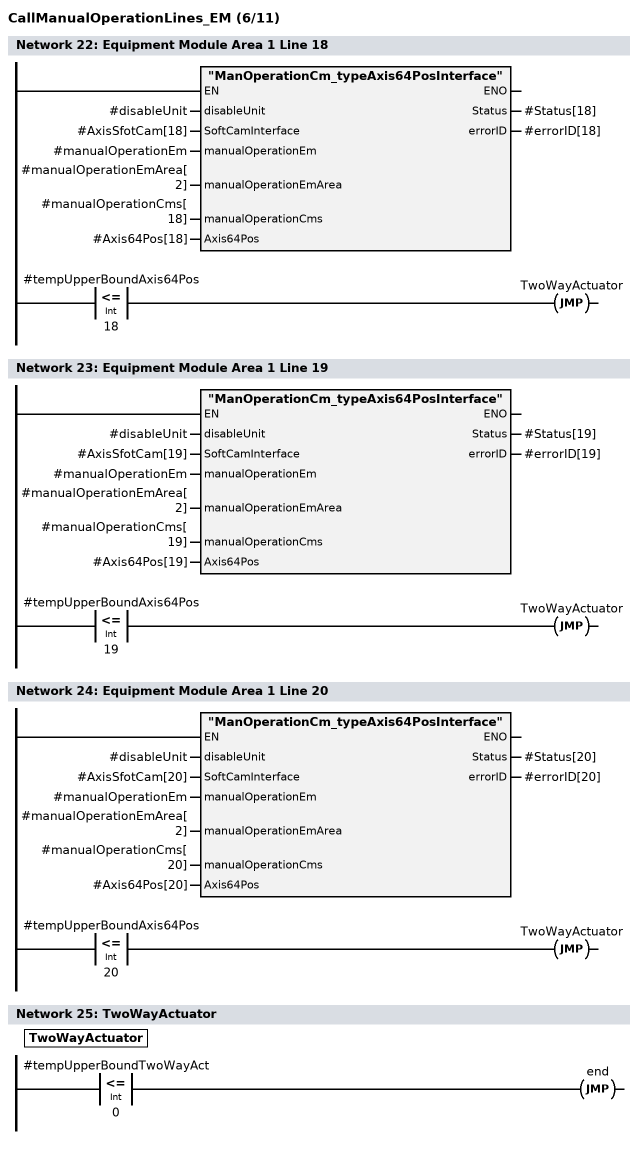
   RUNG wire#powerrail
      "ManOperationCm_typeAxis64PosInterface"(disableUnit := #disableUnit, SoftCamInterface := #AxisSfotCam[18], manualOperationEm := #manualOperationEm, manualOperationEmArea := #manualOperationEmArea[2], manualOperationCms := #manualOperationCms[18], Axis64Pos := #Axis64Pos[18], Status => #Status[18], errorID => #errorID[18])
   END_RUNG
   RUNG wire#powerrail
      { S7_Templates := "SrcType := Int" } LE_Contact(in1 := #tempUpperBoundAxis64Pos, in2 := 18)
      JumpCoil( TwoWayActuator )
   END_RUNG
   // the same network as SCL:
   "ManOperationCm_typeAxis64PosInterface"(disableUnit := #disableUnit,
                           SoftCamInterface := #AxisSfotCam[18],
                           manualOperationEm := #manualOperationEm,
                           manualOperationEmArea := #manualOperationEmArea[2],
                           manualOperationCms := #manualOperationCms[18],
                           Axis64Pos := #Axis64Pos[18],
                           Status => #Status[18],
                           errorID => #errorID[18]);
   IF #tempUpperBoundAxis64Pos <= 18 THEN GOTO TwoWayActuator; END_IF;
END_REGION

REGION Network 23: Equipment Module Area 1 Line 19
   RUNG wire#powerrail
      "ManOperationCm_typeAxis64PosInterface"(disableUnit := #disableUnit, SoftCamInterface := #AxisSfotCam[19], manualOperationEm := #manualOperationEm, manualOperationEmArea := #manualOperationEmArea[2], manualOperationCms := #manualOperationCms[19], Axis64Pos := #Axis64Pos[19], Status => #Status[19], errorID => #errorID[19])
   END_RUNG
   RUNG wire#powerrail
      { S7_Templates := "SrcType := Int" } LE_Contact(in1 := #tempUpperBoundAxis64Pos, in2 := 19)
      JumpCoil( TwoWayActuator )
   END_RUNG
   // the same network as SCL:
   "ManOperationCm_typeAxis64PosInterface"(disableUnit := #disableUnit,
                           SoftCamInterface := #AxisSfotCam[19],
                           manualOperationEm := #manualOperationEm,
                           manualOperationEmArea := #manualOperationEmArea[2],
                           manualOperationCms := #manualOperationCms[19],
                           Axis64Pos := #Axis64Pos[19],
                           Status => #Status[19],
                           errorID => #errorID[19]);
   IF #tempUpperBoundAxis64Pos <= 19 THEN GOTO TwoWayActuator; END_IF;
END_REGION

REGION Network 24: Equipment Module Area 1 Line 20
   RUNG wire#powerrail
      "ManOperationCm_typeAxis64PosInterface"(disableUnit := #disableUnit, SoftCamInterface := #AxisSfotCam[20], manualOperationEm := #manualOperationEm, manualOperationEmArea := #manualOperationEmArea[2], manualOperationCms := #manualOperationCms[20], Axis64Pos := #Axis64Pos[20], Status => #Status[20], errorID => #errorID[20])
   END_RUNG
   RUNG wire#powerrail
      { S7_Templates := "SrcType := Int" } LE_Contact(in1 := #tempUpperBoundAxis64Pos, in2 := 20)
      JumpCoil( TwoWayActuator )
   END_RUNG
   // the same network as SCL:
   "ManOperationCm_typeAxis64PosInterface"(disableUnit := #disableUnit,
                           SoftCamInterface := #AxisSfotCam[20],
                           manualOperationEm := #manualOperationEm,
                           manualOperationEmArea := #manualOperationEmArea[2],
                           manualOperationCms := #manualOperationCms[20],
                           Axis64Pos := #Axis64Pos[20],
                           Status => #Status[20],
                           errorID => #errorID[20]);
   IF #tempUpperBoundAxis64Pos <= 20 THEN GOTO TwoWayActuator; END_IF;
END_REGION

REGION Network 25: TwoWayActuator
   Label( TwoWayActuator )
   RUNG wire#powerrail
      { S7_Templates := "SrcType := Int" } LE_Contact(in1 := #tempUpperBoundTwoWayAct, in2 := 0)
      JumpCoil( end )
   END_RUNG
   // the same network as SCL:
   TwoWayActuator:
   IF #tempUpperBoundTwoWayAct <= 0 THEN GOTO end; END_IF;
END_REGION

REGION Network 26: Equipment Module Area 2 Line 21
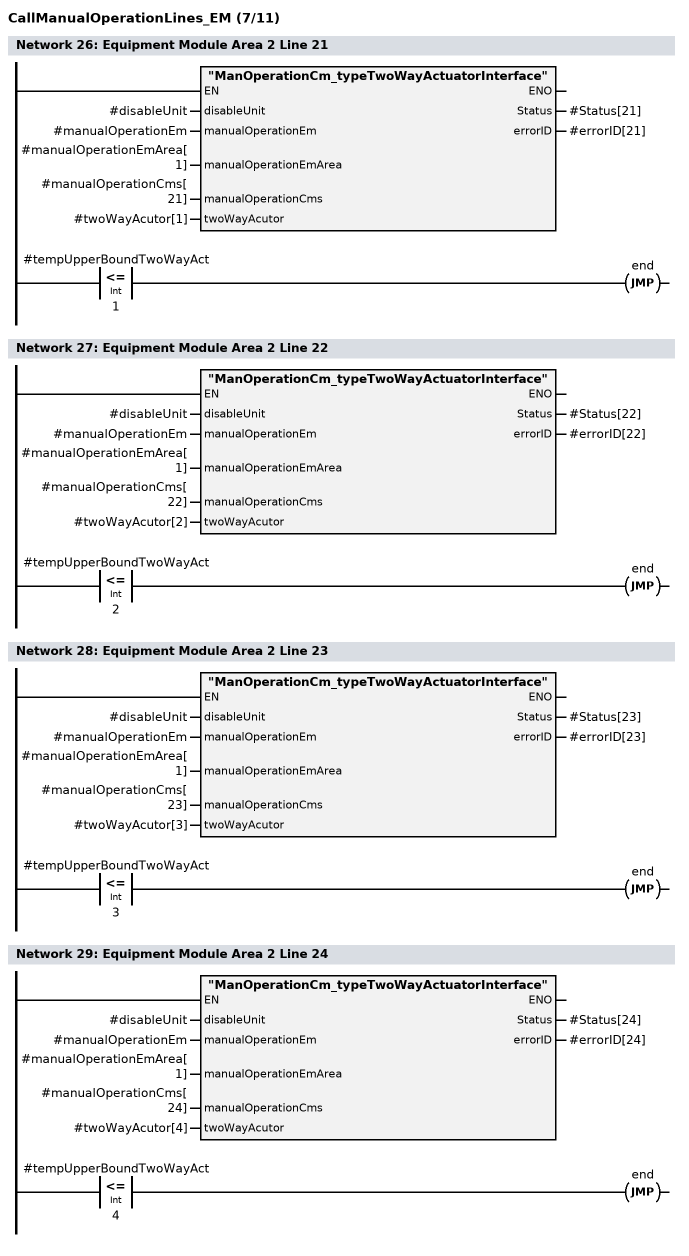
   RUNG wire#powerrail
      "ManOperationCm_typeTwoWayActuatorInterface"(disableUnit := #disableUnit, manualOperationEm := #manualOperationEm, manualOperationEmArea := #manualOperationEmArea[1], manualOperationCms := #manualOperationCms[21], twoWayAcutor := #twoWayAcutor[1], Status => #Status[21], errorID => #errorID[21])
   END_RUNG
   RUNG wire#powerrail
      { S7_Templates := "SrcType := Int" } LE_Contact(in1 := #tempUpperBoundTwoWayAct, in2 := 1)
      JumpCoil( end )
   END_RUNG
   // the same network as SCL:
   "ManOperationCm_typeTwoWayActuatorInterface"(disableUnit := #disableUnit,
                           manualOperationEm := #manualOperationEm,
                           manualOperationEmArea := #manualOperationEmArea[1],
                           manualOperationCms := #manualOperationCms[21],
                           twoWayAcutor := #twoWayAcutor[1],
                           Status => #Status[21],
                           errorID => #errorID[21]);
   IF #tempUpperBoundTwoWayAct <= 1 THEN GOTO end; END_IF;
END_REGION

REGION Network 27: Equipment Module Area 2 Line 22
   RUNG wire#powerrail
      "ManOperationCm_typeTwoWayActuatorInterface"(disableUnit := #disableUnit, manualOperationEm := #manualOperationEm, manualOperationEmArea := #manualOperationEmArea[1], manualOperationCms := #manualOperationCms[22], twoWayAcutor := #twoWayAcutor[2], Status => #Status[22], errorID => #errorID[22])
   END_RUNG
   RUNG wire#powerrail
      { S7_Templates := "SrcType := Int" } LE_Contact(in1 := #tempUpperBoundTwoWayAct, in2 := 2)
      JumpCoil( end )
   END_RUNG
   // the same network as SCL:
   "ManOperationCm_typeTwoWayActuatorInterface"(disableUnit := #disableUnit,
                           manualOperationEm := #manualOperationEm,
                           manualOperationEmArea := #manualOperationEmArea[1],
                           manualOperationCms := #manualOperationCms[22],
                           twoWayAcutor := #twoWayAcutor[2],
                           Status => #Status[22],
                           errorID => #errorID[22]);
   IF #tempUpperBoundTwoWayAct <= 2 THEN GOTO end; END_IF;
END_REGION

REGION Network 28: Equipment Module Area 2 Line 23
   RUNG wire#powerrail
      "ManOperationCm_typeTwoWayActuatorInterface"(disableUnit := #disableUnit, manualOperationEm := #manualOperationEm, manualOperationEmArea := #manualOperationEmArea[1], manualOperationCms := #manualOperationCms[23], twoWayAcutor := #twoWayAcutor[3], Status => #Status[23], errorID => #errorID[23])
   END_RUNG
   RUNG wire#powerrail
      { S7_Templates := "SrcType := Int" } LE_Contact(in1 := #tempUpperBoundTwoWayAct, in2 := 3)
      JumpCoil( end )
   END_RUNG
   // the same network as SCL:
   "ManOperationCm_typeTwoWayActuatorInterface"(disableUnit := #disableUnit,
                           manualOperationEm := #manualOperationEm,
                           manualOperationEmArea := #manualOperationEmArea[1],
                           manualOperationCms := #manualOperationCms[23],
                           twoWayAcutor := #twoWayAcutor[3],
                           Status => #Status[23],
                           errorID => #errorID[23]);
   IF #tempUpperBoundTwoWayAct <= 3 THEN GOTO end; END_IF;
END_REGION

REGION Network 29: Equipment Module Area 2 Line 24
   RUNG wire#powerrail
      "ManOperationCm_typeTwoWayActuatorInterface"(disableUnit := #disableUnit, manualOperationEm := #manualOperationEm, manualOperationEmArea := #manualOperationEmArea[1], manualOperationCms := #manualOperationCms[24], twoWayAcutor := #twoWayAcutor[4], Status => #Status[24], errorID => #errorID[24])
   END_RUNG
   RUNG wire#powerrail
      { S7_Templates := "SrcType := Int" } LE_Contact(in1 := #tempUpperBoundTwoWayAct, in2 := 4)
      JumpCoil( end )
   END_RUNG
   // the same network as SCL:
   "ManOperationCm_typeTwoWayActuatorInterface"(disableUnit := #disableUnit,
                           manualOperationEm := #manualOperationEm,
                           manualOperationEmArea := #manualOperationEmArea[1],
                           manualOperationCms := #manualOperationCms[24],
                           twoWayAcutor := #twoWayAcutor[4],
                           Status => #Status[24],
                           errorID => #errorID[24]);
   IF #tempUpperBoundTwoWayAct <= 4 THEN GOTO end; END_IF;
END_REGION

REGION Network 30: Equipment Module Area 2 Line 25
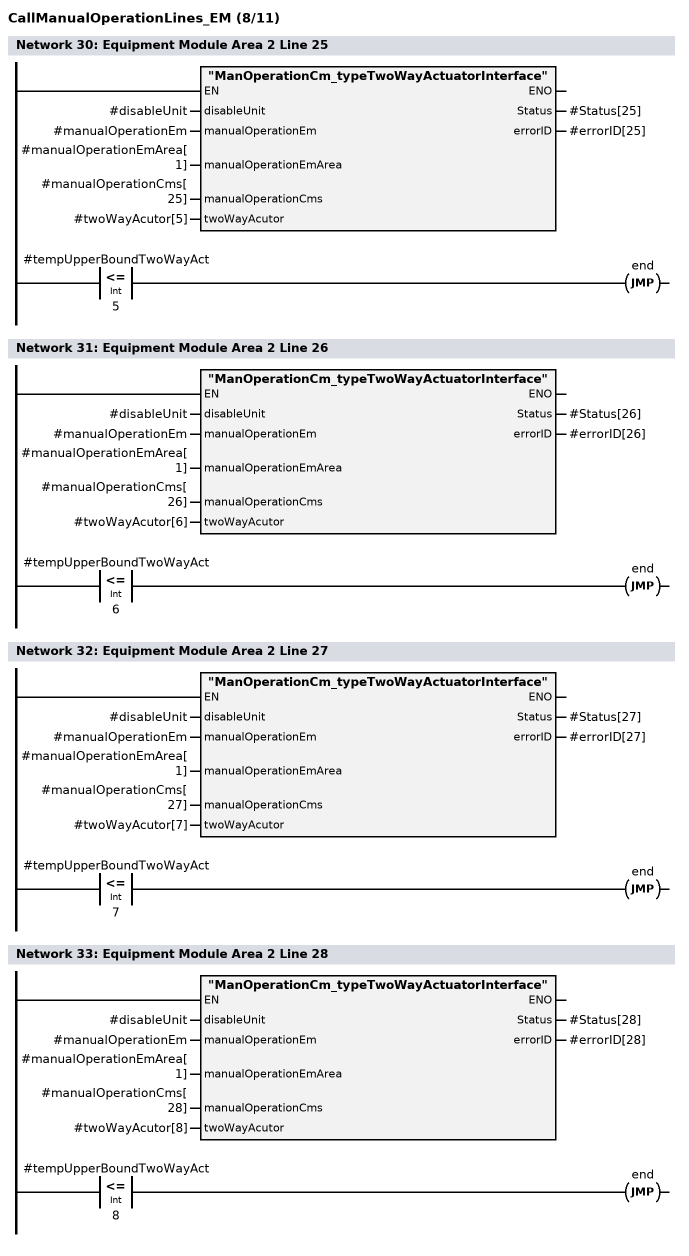
   RUNG wire#powerrail
      "ManOperationCm_typeTwoWayActuatorInterface"(disableUnit := #disableUnit, manualOperationEm := #manualOperationEm, manualOperationEmArea := #manualOperationEmArea[1], manualOperationCms := #manualOperationCms[25], twoWayAcutor := #twoWayAcutor[5], Status => #Status[25], errorID => #errorID[25])
   END_RUNG
   RUNG wire#powerrail
      { S7_Templates := "SrcType := Int" } LE_Contact(in1 := #tempUpperBoundTwoWayAct, in2 := 5)
      JumpCoil( end )
   END_RUNG
   // the same network as SCL:
   "ManOperationCm_typeTwoWayActuatorInterface"(disableUnit := #disableUnit,
                           manualOperationEm := #manualOperationEm,
                           manualOperationEmArea := #manualOperationEmArea[1],
                           manualOperationCms := #manualOperationCms[25],
                           twoWayAcutor := #twoWayAcutor[5],
                           Status => #Status[25],
                           errorID => #errorID[25]);
   IF #tempUpperBoundTwoWayAct <= 5 THEN GOTO end; END_IF;
END_REGION

REGION Network 31: Equipment Module Area 2 Line 26
   RUNG wire#powerrail
      "ManOperationCm_typeTwoWayActuatorInterface"(disableUnit := #disableUnit, manualOperationEm := #manualOperationEm, manualOperationEmArea := #manualOperationEmArea[1], manualOperationCms := #manualOperationCms[26], twoWayAcutor := #twoWayAcutor[6], Status => #Status[26], errorID => #errorID[26])
   END_RUNG
   RUNG wire#powerrail
      { S7_Templates := "SrcType := Int" } LE_Contact(in1 := #tempUpperBoundTwoWayAct, in2 := 6)
      JumpCoil( end )
   END_RUNG
   // the same network as SCL:
   "ManOperationCm_typeTwoWayActuatorInterface"(disableUnit := #disableUnit,
                           manualOperationEm := #manualOperationEm,
                           manualOperationEmArea := #manualOperationEmArea[1],
                           manualOperationCms := #manualOperationCms[26],
                           twoWayAcutor := #twoWayAcutor[6],
                           Status => #Status[26],
                           errorID => #errorID[26]);
   IF #tempUpperBoundTwoWayAct <= 6 THEN GOTO end; END_IF;
END_REGION

REGION Network 32: Equipment Module Area 2 Line 27
   RUNG wire#powerrail
      "ManOperationCm_typeTwoWayActuatorInterface"(disableUnit := #disableUnit, manualOperationEm := #manualOperationEm, manualOperationEmArea := #manualOperationEmArea[1], manualOperationCms := #manualOperationCms[27], twoWayAcutor := #twoWayAcutor[7], Status => #Status[27], errorID => #errorID[27])
   END_RUNG
   RUNG wire#powerrail
      { S7_Templates := "SrcType := Int" } LE_Contact(in1 := #tempUpperBoundTwoWayAct, in2 := 7)
      JumpCoil( end )
   END_RUNG
   // the same network as SCL:
   "ManOperationCm_typeTwoWayActuatorInterface"(disableUnit := #disableUnit,
                           manualOperationEm := #manualOperationEm,
                           manualOperationEmArea := #manualOperationEmArea[1],
                           manualOperationCms := #manualOperationCms[27],
                           twoWayAcutor := #twoWayAcutor[7],
                           Status => #Status[27],
                           errorID => #errorID[27]);
   IF #tempUpperBoundTwoWayAct <= 7 THEN GOTO end; END_IF;
END_REGION

REGION Network 33: Equipment Module Area 2 Line 28
   RUNG wire#powerrail
      "ManOperationCm_typeTwoWayActuatorInterface"(disableUnit := #disableUnit, manualOperationEm := #manualOperationEm, manualOperationEmArea := #manualOperationEmArea[1], manualOperationCms := #manualOperationCms[28], twoWayAcutor := #twoWayAcutor[8], Status => #Status[28], errorID => #errorID[28])
   END_RUNG
   RUNG wire#powerrail
      { S7_Templates := "SrcType := Int" } LE_Contact(in1 := #tempUpperBoundTwoWayAct, in2 := 8)
      JumpCoil( end )
   END_RUNG
   // the same network as SCL:
   "ManOperationCm_typeTwoWayActuatorInterface"(disableUnit := #disableUnit,
                           manualOperationEm := #manualOperationEm,
                           manualOperationEmArea := #manualOperationEmArea[1],
                           manualOperationCms := #manualOperationCms[28],
                           twoWayAcutor := #twoWayAcutor[8],
                           Status => #Status[28],
                           errorID => #errorID[28]);
   IF #tempUpperBoundTwoWayAct <= 8 THEN GOTO end; END_IF;
END_REGION

REGION Network 34: Equipment Module Area 2 Line 29
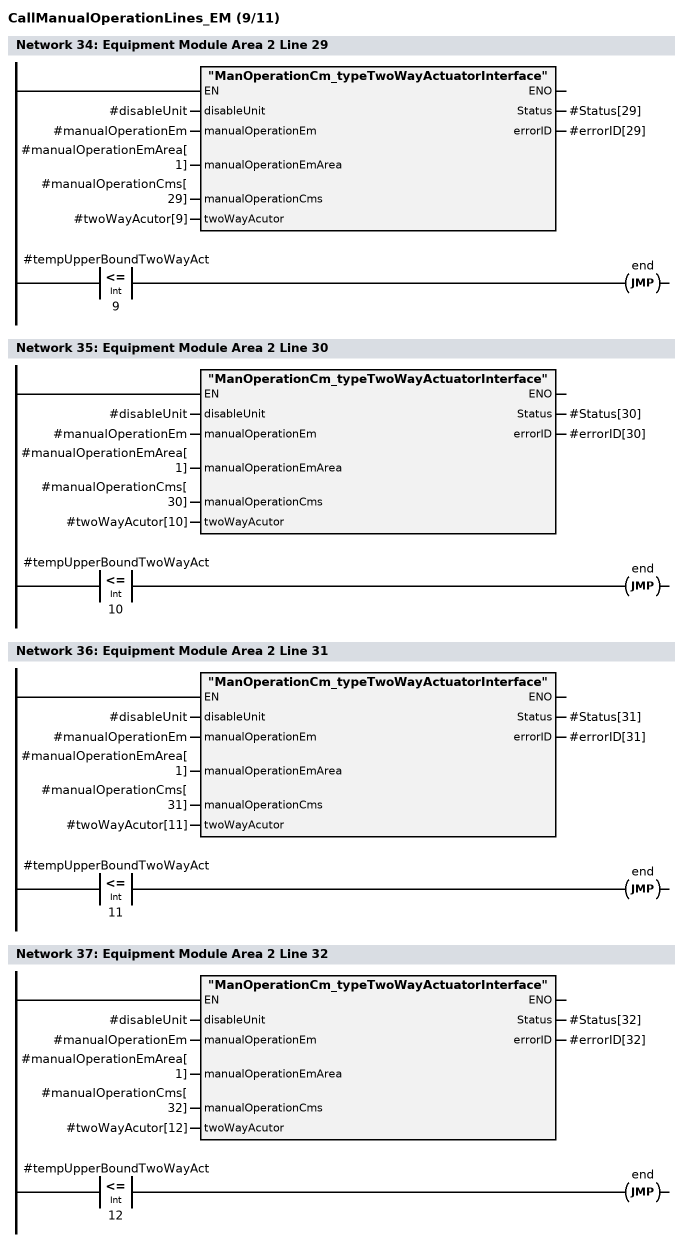
   RUNG wire#powerrail
      "ManOperationCm_typeTwoWayActuatorInterface"(disableUnit := #disableUnit, manualOperationEm := #manualOperationEm, manualOperationEmArea := #manualOperationEmArea[1], manualOperationCms := #manualOperationCms[29], twoWayAcutor := #twoWayAcutor[9], Status => #Status[29], errorID => #errorID[29])
   END_RUNG
   RUNG wire#powerrail
      { S7_Templates := "SrcType := Int" } LE_Contact(in1 := #tempUpperBoundTwoWayAct, in2 := 9)
      JumpCoil( end )
   END_RUNG
   // the same network as SCL:
   "ManOperationCm_typeTwoWayActuatorInterface"(disableUnit := #disableUnit,
                           manualOperationEm := #manualOperationEm,
                           manualOperationEmArea := #manualOperationEmArea[1],
                           manualOperationCms := #manualOperationCms[29],
                           twoWayAcutor := #twoWayAcutor[9],
                           Status => #Status[29],
                           errorID => #errorID[29]);
   IF #tempUpperBoundTwoWayAct <= 9 THEN GOTO end; END_IF;
END_REGION

REGION Network 35: Equipment Module Area 2 Line 30
   RUNG wire#powerrail
      "ManOperationCm_typeTwoWayActuatorInterface"(disableUnit := #disableUnit, manualOperationEm := #manualOperationEm, manualOperationEmArea := #manualOperationEmArea[1], manualOperationCms := #manualOperationCms[30], twoWayAcutor := #twoWayAcutor[10], Status => #Status[30], errorID => #errorID[30])
   END_RUNG
   RUNG wire#powerrail
      { S7_Templates := "SrcType := Int" } LE_Contact(in1 := #tempUpperBoundTwoWayAct, in2 := 10)
      JumpCoil( end )
   END_RUNG
   // the same network as SCL:
   "ManOperationCm_typeTwoWayActuatorInterface"(disableUnit := #disableUnit,
                           manualOperationEm := #manualOperationEm,
                           manualOperationEmArea := #manualOperationEmArea[1],
                           manualOperationCms := #manualOperationCms[30],
                           twoWayAcutor := #twoWayAcutor[10],
                           Status => #Status[30],
                           errorID => #errorID[30]);
   IF #tempUpperBoundTwoWayAct <= 10 THEN GOTO end; END_IF;
END_REGION

REGION Network 36: Equipment Module Area 2 Line 31
   RUNG wire#powerrail
      "ManOperationCm_typeTwoWayActuatorInterface"(disableUnit := #disableUnit, manualOperationEm := #manualOperationEm, manualOperationEmArea := #manualOperationEmArea[1], manualOperationCms := #manualOperationCms[31], twoWayAcutor := #twoWayAcutor[11], Status => #Status[31], errorID => #errorID[31])
   END_RUNG
   RUNG wire#powerrail
      { S7_Templates := "SrcType := Int" } LE_Contact(in1 := #tempUpperBoundTwoWayAct, in2 := 11)
      JumpCoil( end )
   END_RUNG
   // the same network as SCL:
   "ManOperationCm_typeTwoWayActuatorInterface"(disableUnit := #disableUnit,
                           manualOperationEm := #manualOperationEm,
                           manualOperationEmArea := #manualOperationEmArea[1],
                           manualOperationCms := #manualOperationCms[31],
                           twoWayAcutor := #twoWayAcutor[11],
                           Status => #Status[31],
                           errorID => #errorID[31]);
   IF #tempUpperBoundTwoWayAct <= 11 THEN GOTO end; END_IF;
END_REGION

REGION Network 37: Equipment Module Area 2 Line 32
   RUNG wire#powerrail
      "ManOperationCm_typeTwoWayActuatorInterface"(disableUnit := #disableUnit, manualOperationEm := #manualOperationEm, manualOperationEmArea := #manualOperationEmArea[1], manualOperationCms := #manualOperationCms[32], twoWayAcutor := #twoWayAcutor[12], Status => #Status[32], errorID => #errorID[32])
   END_RUNG
   RUNG wire#powerrail
      { S7_Templates := "SrcType := Int" } LE_Contact(in1 := #tempUpperBoundTwoWayAct, in2 := 12)
      JumpCoil( end )
   END_RUNG
   // the same network as SCL:
   "ManOperationCm_typeTwoWayActuatorInterface"(disableUnit := #disableUnit,
                           manualOperationEm := #manualOperationEm,
                           manualOperationEmArea := #manualOperationEmArea[1],
                           manualOperationCms := #manualOperationCms[32],
                           twoWayAcutor := #twoWayAcutor[12],
                           Status => #Status[32],
                           errorID => #errorID[32]);
   IF #tempUpperBoundTwoWayAct <= 12 THEN GOTO end; END_IF;
END_REGION

REGION Network 38: Equipment Module Area 2 Line 33
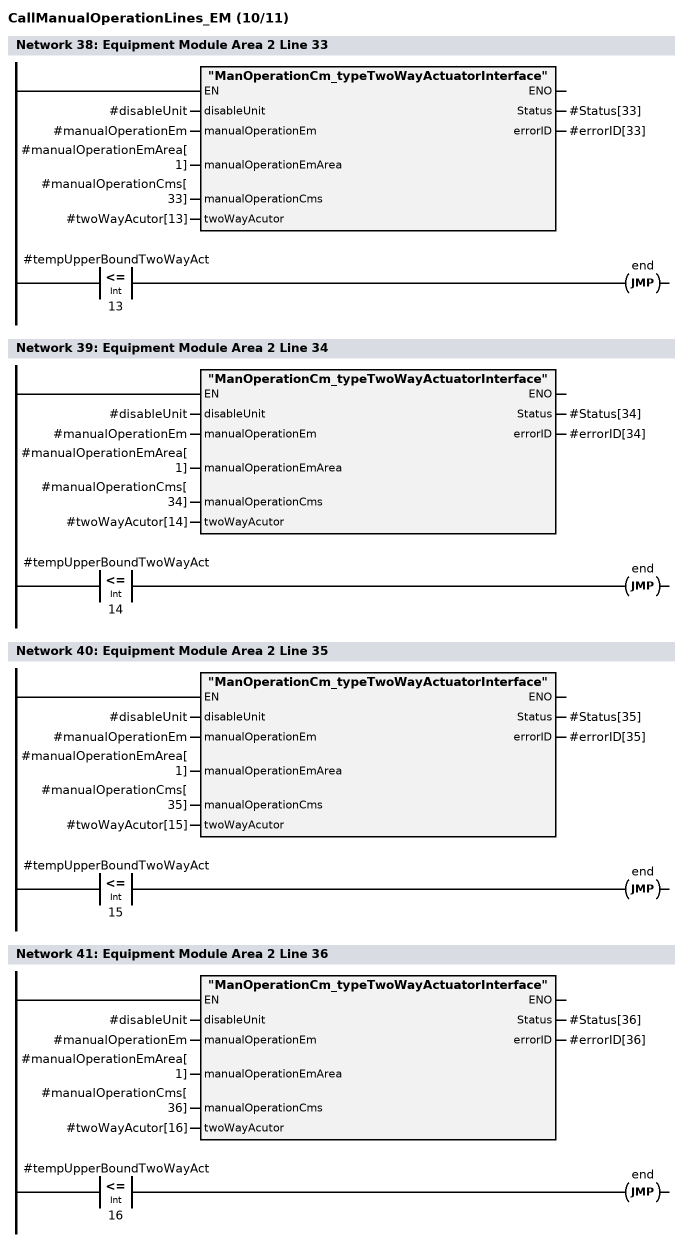
   RUNG wire#powerrail
      "ManOperationCm_typeTwoWayActuatorInterface"(disableUnit := #disableUnit, manualOperationEm := #manualOperationEm, manualOperationEmArea := #manualOperationEmArea[1], manualOperationCms := #manualOperationCms[33], twoWayAcutor := #twoWayAcutor[13], Status => #Status[33], errorID => #errorID[33])
   END_RUNG
   RUNG wire#powerrail
      { S7_Templates := "SrcType := Int" } LE_Contact(in1 := #tempUpperBoundTwoWayAct, in2 := 13)
      JumpCoil( end )
   END_RUNG
   // the same network as SCL:
   "ManOperationCm_typeTwoWayActuatorInterface"(disableUnit := #disableUnit,
                           manualOperationEm := #manualOperationEm,
                           manualOperationEmArea := #manualOperationEmArea[1],
                           manualOperationCms := #manualOperationCms[33],
                           twoWayAcutor := #twoWayAcutor[13],
                           Status => #Status[33],
                           errorID => #errorID[33]);
   IF #tempUpperBoundTwoWayAct <= 13 THEN GOTO end; END_IF;
END_REGION

REGION Network 39: Equipment Module Area 2 Line 34
   RUNG wire#powerrail
      "ManOperationCm_typeTwoWayActuatorInterface"(disableUnit := #disableUnit, manualOperationEm := #manualOperationEm, manualOperationEmArea := #manualOperationEmArea[1], manualOperationCms := #manualOperationCms[34], twoWayAcutor := #twoWayAcutor[14], Status => #Status[34], errorID => #errorID[34])
   END_RUNG
   RUNG wire#powerrail
      { S7_Templates := "SrcType := Int" } LE_Contact(in1 := #tempUpperBoundTwoWayAct, in2 := 14)
      JumpCoil( end )
   END_RUNG
   // the same network as SCL:
   "ManOperationCm_typeTwoWayActuatorInterface"(disableUnit := #disableUnit,
                           manualOperationEm := #manualOperationEm,
                           manualOperationEmArea := #manualOperationEmArea[1],
                           manualOperationCms := #manualOperationCms[34],
                           twoWayAcutor := #twoWayAcutor[14],
                           Status => #Status[34],
                           errorID => #errorID[34]);
   IF #tempUpperBoundTwoWayAct <= 14 THEN GOTO end; END_IF;
END_REGION

REGION Network 40: Equipment Module Area 2 Line 35
   RUNG wire#powerrail
      "ManOperationCm_typeTwoWayActuatorInterface"(disableUnit := #disableUnit, manualOperationEm := #manualOperationEm, manualOperationEmArea := #manualOperationEmArea[1], manualOperationCms := #manualOperationCms[35], twoWayAcutor := #twoWayAcutor[15], Status => #Status[35], errorID => #errorID[35])
   END_RUNG
   RUNG wire#powerrail
      { S7_Templates := "SrcType := Int" } LE_Contact(in1 := #tempUpperBoundTwoWayAct, in2 := 15)
      JumpCoil( end )
   END_RUNG
   // the same network as SCL:
   "ManOperationCm_typeTwoWayActuatorInterface"(disableUnit := #disableUnit,
                           manualOperationEm := #manualOperationEm,
                           manualOperationEmArea := #manualOperationEmArea[1],
                           manualOperationCms := #manualOperationCms[35],
                           twoWayAcutor := #twoWayAcutor[15],
                           Status => #Status[35],
                           errorID => #errorID[35]);
   IF #tempUpperBoundTwoWayAct <= 15 THEN GOTO end; END_IF;
END_REGION

REGION Network 41: Equipment Module Area 2 Line 36
   RUNG wire#powerrail
      "ManOperationCm_typeTwoWayActuatorInterface"(disableUnit := #disableUnit, manualOperationEm := #manualOperationEm, manualOperationEmArea := #manualOperationEmArea[1], manualOperationCms := #manualOperationCms[36], twoWayAcutor := #twoWayAcutor[16], Status => #Status[36], errorID => #errorID[36])
   END_RUNG
   RUNG wire#powerrail
      { S7_Templates := "SrcType := Int" } LE_Contact(in1 := #tempUpperBoundTwoWayAct, in2 := 16)
      JumpCoil( end )
   END_RUNG
   // the same network as SCL:
   "ManOperationCm_typeTwoWayActuatorInterface"(disableUnit := #disableUnit,
                           manualOperationEm := #manualOperationEm,
                           manualOperationEmArea := #manualOperationEmArea[1],
                           manualOperationCms := #manualOperationCms[36],
                           twoWayAcutor := #twoWayAcutor[16],
                           Status => #Status[36],
                           errorID => #errorID[36]);
   IF #tempUpperBoundTwoWayAct <= 16 THEN GOTO end; END_IF;
END_REGION

REGION Network 42: Equipment Module Area 2 Line 37
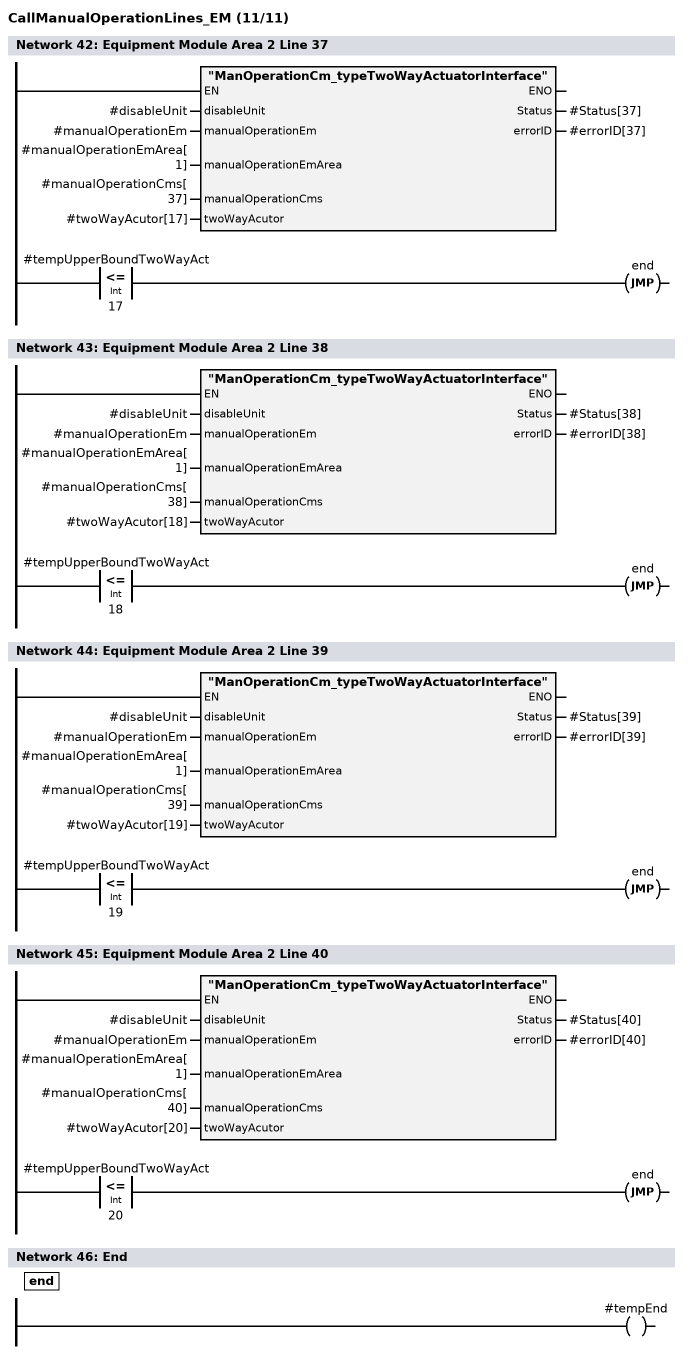
   RUNG wire#powerrail
      "ManOperationCm_typeTwoWayActuatorInterface"(disableUnit := #disableUnit, manualOperationEm := #manualOperationEm, manualOperationEmArea := #manualOperationEmArea[1], manualOperationCms := #manualOperationCms[37], twoWayAcutor := #twoWayAcutor[17], Status => #Status[37], errorID => #errorID[37])
   END_RUNG
   RUNG wire#powerrail
      { S7_Templates := "SrcType := Int" } LE_Contact(in1 := #tempUpperBoundTwoWayAct, in2 := 17)
      JumpCoil( end )
   END_RUNG
   // the same network as SCL:
   "ManOperationCm_typeTwoWayActuatorInterface"(disableUnit := #disableUnit,
                           manualOperationEm := #manualOperationEm,
                           manualOperationEmArea := #manualOperationEmArea[1],
                           manualOperationCms := #manualOperationCms[37],
                           twoWayAcutor := #twoWayAcutor[17],
                           Status => #Status[37],
                           errorID => #errorID[37]);
   IF #tempUpperBoundTwoWayAct <= 17 THEN GOTO end; END_IF;
END_REGION

REGION Network 43: Equipment Module Area 2 Line 38
   RUNG wire#powerrail
      "ManOperationCm_typeTwoWayActuatorInterface"(disableUnit := #disableUnit, manualOperationEm := #manualOperationEm, manualOperationEmArea := #manualOperationEmArea[1], manualOperationCms := #manualOperationCms[38], twoWayAcutor := #twoWayAcutor[18], Status => #Status[38], errorID => #errorID[38])
   END_RUNG
   RUNG wire#powerrail
      { S7_Templates := "SrcType := Int" } LE_Contact(in1 := #tempUpperBoundTwoWayAct, in2 := 18)
      JumpCoil( end )
   END_RUNG
   // the same network as SCL:
   "ManOperationCm_typeTwoWayActuatorInterface"(disableUnit := #disableUnit,
                           manualOperationEm := #manualOperationEm,
                           manualOperationEmArea := #manualOperationEmArea[1],
                           manualOperationCms := #manualOperationCms[38],
                           twoWayAcutor := #twoWayAcutor[18],
                           Status => #Status[38],
                           errorID => #errorID[38]);
   IF #tempUpperBoundTwoWayAct <= 18 THEN GOTO end; END_IF;
END_REGION

REGION Network 44: Equipment Module Area 2 Line 39
   RUNG wire#powerrail
      "ManOperationCm_typeTwoWayActuatorInterface"(disableUnit := #disableUnit, manualOperationEm := #manualOperationEm, manualOperationEmArea := #manualOperationEmArea[1], manualOperationCms := #manualOperationCms[39], twoWayAcutor := #twoWayAcutor[19], Status => #Status[39], errorID => #errorID[39])
   END_RUNG
   RUNG wire#powerrail
      { S7_Templates := "SrcType := Int" } LE_Contact(in1 := #tempUpperBoundTwoWayAct, in2 := 19)
      JumpCoil( end )
   END_RUNG
   // the same network as SCL:
   "ManOperationCm_typeTwoWayActuatorInterface"(disableUnit := #disableUnit,
                           manualOperationEm := #manualOperationEm,
                           manualOperationEmArea := #manualOperationEmArea[1],
                           manualOperationCms := #manualOperationCms[39],
                           twoWayAcutor := #twoWayAcutor[19],
                           Status => #Status[39],
                           errorID => #errorID[39]);
   IF #tempUpperBoundTwoWayAct <= 19 THEN GOTO end; END_IF;
END_REGION

REGION Network 45: Equipment Module Area 2 Line 40
   RUNG wire#powerrail
      "ManOperationCm_typeTwoWayActuatorInterface"(disableUnit := #disableUnit, manualOperationEm := #manualOperationEm, manualOperationEmArea := #manualOperationEmArea[1], manualOperationCms := #manualOperationCms[40], twoWayAcutor := #twoWayAcutor[20], Status => #Status[40], errorID => #errorID[40])
   END_RUNG
   RUNG wire#powerrail
      { S7_Templates := "SrcType := Int" } LE_Contact(in1 := #tempUpperBoundTwoWayAct, in2 := 20)
      JumpCoil( end )
   END_RUNG
   // the same network as SCL:
   "ManOperationCm_typeTwoWayActuatorInterface"(disableUnit := #disableUnit,
                           manualOperationEm := #manualOperationEm,
                           manualOperationEmArea := #manualOperationEmArea[1],
                           manualOperationCms := #manualOperationCms[40],
                           twoWayAcutor := #twoWayAcutor[20],
                           Status => #Status[40],
                           errorID => #errorID[40]);
   IF #tempUpperBoundTwoWayAct <= 20 THEN GOTO end; END_IF;
END_REGION

REGION Network 46: End
   Label( end )
   RUNG wire#powerrail
      Coil( #tempEnd )
   END_RUNG
   // the same network as SCL:
   end:
   #tempEnd := TRUE;
END_REGION
END_FUNCTION

FUNCTION "ManOperationCm_typeAxisControlInterface" : Void   // FC76, LAD
// stored: SetENOAutomatically false
   VAR_INPUT
      disableUnit : Bool;
   END_VAR
   VAR_OUTPUT
      Status : Word;
      errorID : Word;
   END_VAR
   VAR_IN_OUT
      manualOperationEm : "LAF_typeManEm";
      manualOperationEmArea : "LAF_typeManOperationArea";
      manualOperationCms : "LAF_typeManOperation";
      Axis : "LBC_typeAxisControlInterface";
   END_VAR
BEGIN

REGION Network 1: Manual Operation Cm - typeAxisControlInterface
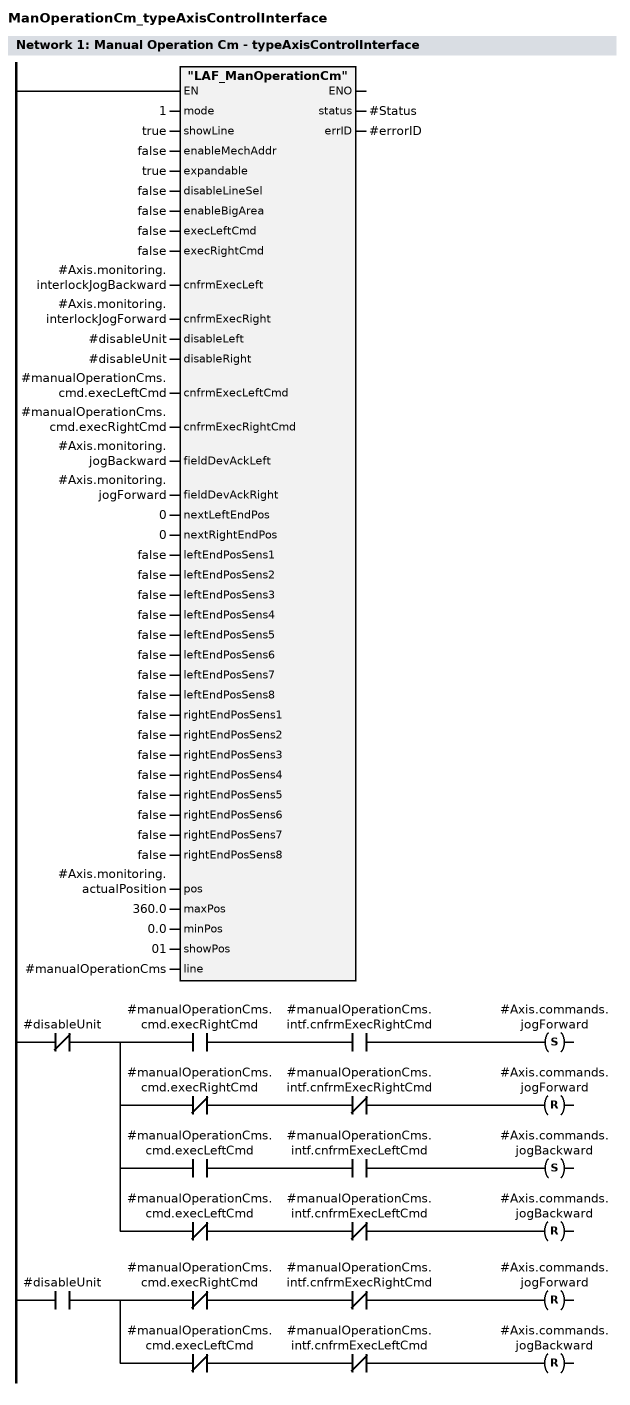
   RUNG wire#powerrail
      "LAF_ManOperationCm"(mode := 1, showLine := true, enableMechAddr := false, expandable := true, disableLineSel := false, enableBigArea := false, execLeftCmd := false, execRightCmd := false, cnfrmExecLeft := #Axis.monitoring.interlockJogBackward, cnfrmExecRight := #Axis.monitoring.interlockJogForward, disableLeft := #disableUnit, disableRight := #disableUnit, cnfrmExecLeftCmd := #manualOperationCms.cmd.execLeftCmd, cnfrmExecRightCmd := #manualOperationCms.cmd.execRightCmd, fieldDevAckLeft := #Axis.monitoring.jogBackward, fieldDevAckRight := #Axis.monitoring.jogForward, nextLeftEndPos := 0, nextRightEndPos := 0, leftEndPosSens1 := false, leftEndPosSens2 := false, leftEndPosSens3 := false, leftEndPosSens4 := false, leftEndPosSens5 := false, leftEndPosSens6 := false, leftEndPosSens7 := false, leftEndPosSens8 := false, rightEndPosSens1 := false, rightEndPosSens2 := false, rightEndPosSens3 := false, rightEndPosSens4 := false, rightEndPosSens5 := false, rightEndPosSens6 := false, rightEndPosSens7 := false, rightEndPosSens8 := false, pos := #Axis.monitoring.actualPosition, maxPos := 360.0, minPos := 0.0, showPos := 01, line := #manualOperationCms, status => #Status, errID => #errorID)
   END_RUNG
   RUNG wire#powerrail
      I_Contact( #disableUnit )
      wire#w1
      Contact( #manualOperationCms.cmd.execRightCmd )
      Contact( #manualOperationCms.intf.cnfrmExecRightCmd )
      S_Coil( #Axis.commands.jogForward )
   END_RUNG
   RUNG wire#w1
      I_Contact( #manualOperationCms.cmd.execRightCmd )
      I_Contact( #manualOperationCms.intf.cnfrmExecRightCmd )
      R_Coil( #Axis.commands.jogForward )
   END_RUNG
   RUNG wire#w1
      Contact( #manualOperationCms.cmd.execLeftCmd )
      Contact( #manualOperationCms.intf.cnfrmExecLeftCmd )
      S_Coil( #Axis.commands.jogBackward )
   END_RUNG
   RUNG wire#w1
      I_Contact( #manualOperationCms.cmd.execLeftCmd )
      I_Contact( #manualOperationCms.intf.cnfrmExecLeftCmd )
      R_Coil( #Axis.commands.jogBackward )
   END_RUNG
   RUNG wire#powerrail
      Contact( #disableUnit )
      wire#w2
      I_Contact( #manualOperationCms.cmd.execRightCmd )
      I_Contact( #manualOperationCms.intf.cnfrmExecRightCmd )
      R_Coil( #Axis.commands.jogForward )
   END_RUNG
   RUNG wire#w2
      I_Contact( #manualOperationCms.cmd.execLeftCmd )
      I_Contact( #manualOperationCms.intf.cnfrmExecLeftCmd )
      R_Coil( #Axis.commands.jogBackward )
   END_RUNG
   // the same network as SCL:
   "LAF_ManOperationCm"(mode := 1,
                        showLine := true,
                        enableMechAddr := false,
                        expandable := true,
                        disableLineSel := false,
                        enableBigArea := false,
                        execLeftCmd := false,
                        execRightCmd := false,
                        cnfrmExecLeft := #Axis.monitoring.interlockJogBackward,
                        cnfrmExecRight := #Axis.monitoring.interlockJogForward,
                        disableLeft := #disableUnit,
                        disableRight := #disableUnit,
                        cnfrmExecLeftCmd := #manualOperationCms.cmd.execLeftCmd,
                        cnfrmExecRightCmd := #manualOperationCms.cmd.execRightCmd,
                        fieldDevAckLeft := #Axis.monitoring.jogBackward,
                        fieldDevAckRight := #Axis.monitoring.jogForward,
                        nextLeftEndPos := 0,
                        nextRightEndPos := 0,
                        leftEndPosSens1 := false,
                        leftEndPosSens2 := false,
                        leftEndPosSens3 := false,
                        leftEndPosSens4 := false,
                        leftEndPosSens5 := false,
                        leftEndPosSens6 := false,
                        leftEndPosSens7 := false,
                        leftEndPosSens8 := false,
                        rightEndPosSens1 := false,
                        rightEndPosSens2 := false,
                        rightEndPosSens3 := false,
                        rightEndPosSens4 := false,
                        rightEndPosSens5 := false,
                        rightEndPosSens6 := false,
                        rightEndPosSens7 := false,
                        rightEndPosSens8 := false,
                        pos := #Axis.monitoring.actualPosition,
                        maxPos := 360.0,
                        minPos := 0.0,
                        showPos := 01,
                        line := #manualOperationCms,
                        status => #Status,
                        errID => #errorID);
   IF NOT #disableUnit AND #manualOperationCms.cmd.execRightCmd AND #manualOperationCms.intf.cnfrmExecRightCmd THEN
       #Axis.commands.jogForward := TRUE;
   END_IF;
   IF NOT #disableUnit AND NOT #manualOperationCms.cmd.execRightCmd AND NOT #manualOperationCms.intf.cnfrmExecRightCmd THEN
       #Axis.commands.jogForward := FALSE;
   END_IF;
   IF NOT #disableUnit AND #manualOperationCms.cmd.execLeftCmd AND #manualOperationCms.intf.cnfrmExecLeftCmd THEN
       #Axis.commands.jogBackward := TRUE;
   END_IF;
   IF NOT #disableUnit AND NOT #manualOperationCms.cmd.execLeftCmd AND NOT #manualOperationCms.intf.cnfrmExecLeftCmd THEN
       #Axis.commands.jogBackward := FALSE;
   END_IF;
   IF #disableUnit AND NOT #manualOperationCms.cmd.execRightCmd AND NOT #manualOperationCms.intf.cnfrmExecRightCmd THEN
       #Axis.commands.jogForward := FALSE;
   END_IF;
   IF #disableUnit AND NOT #manualOperationCms.cmd.execLeftCmd AND NOT #manualOperationCms.intf.cnfrmExecLeftCmd THEN
       #Axis.commands.jogBackward := FALSE;
   END_IF;
END_REGION
END_FUNCTION

FUNCTION "ManOperationCm_typeAxis64PosInterface" : Void   // FC80, LAD
// stored: SetENOAutomatically false
   VAR_INPUT
      disableUnit : Bool;
      SoftCamInterface : "LER_typeSoftCamRelation";
   END_VAR
   VAR_OUTPUT
      Status : Word;
      errorID : Word;
   END_VAR
   VAR_IN_OUT
      manualOperationEm : "LAF_typeManEm";
      manualOperationEmArea : "LAF_typeManOperationArea";
      manualOperationCms : "LAF_typeManOperation";
      Axis64Pos : "LBC_typeAxis64PosInterface";
   END_VAR
   VAR_TEMP
      tempMaxPos : LReal;
      tempIndex : Int;
   END_VAR
BEGIN

REGION Network 1 (SCL): MaxPos Find
   FOR #tempIndex := 0 TO 15 DO
       IF #Axis64Pos.configuration.setPositions[#tempIndex].position > #tempMaxPos THEN
           #tempMaxPos := #Axis64Pos.configuration.setPositions[#tempIndex].position;
       END_IF;
   END_FOR;
END_REGION

REGION Network 2: Manual Operation Cm - typeAxis64PosInterface
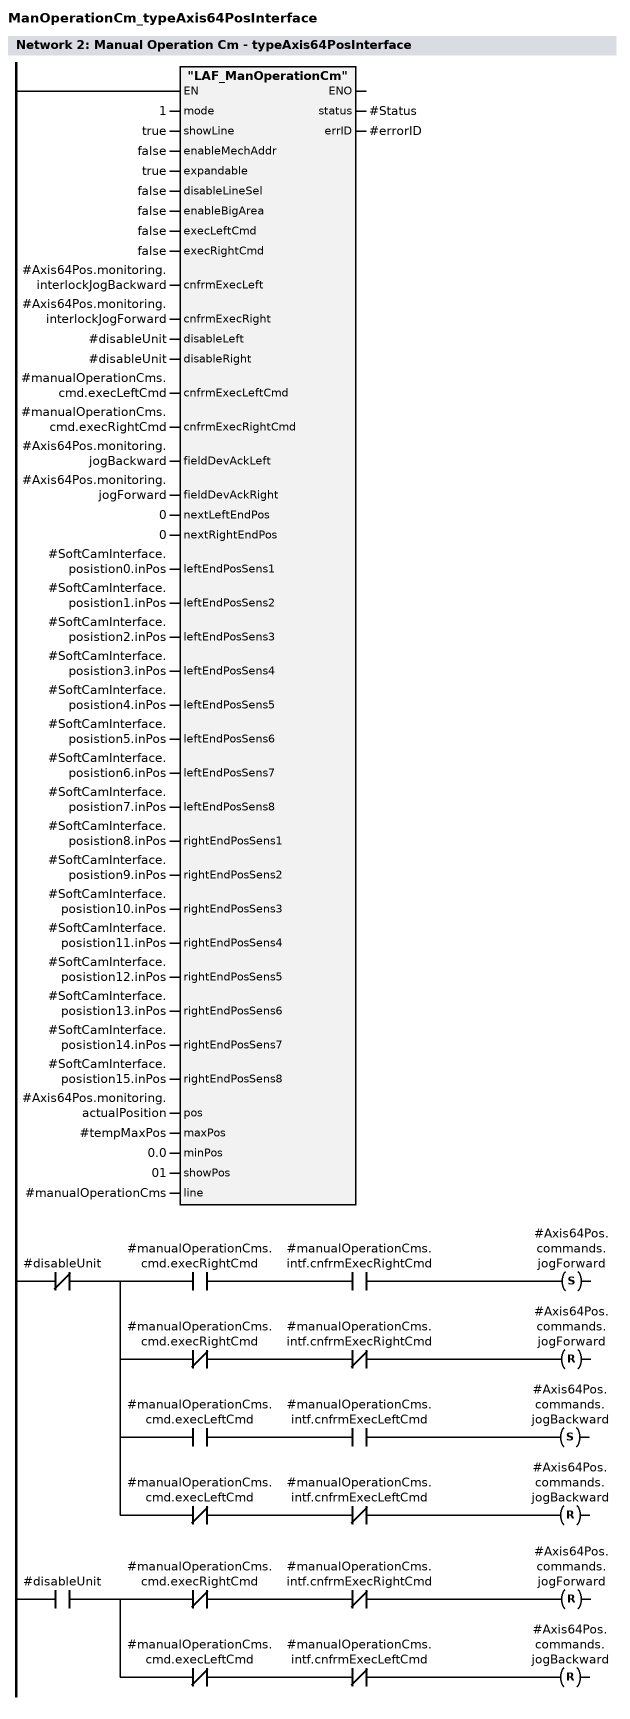
   RUNG wire#powerrail
      "LAF_ManOperationCm"(mode := 1, showLine := true, enableMechAddr := false, expandable := true, disableLineSel := false, enableBigArea := false, execLeftCmd := false, execRightCmd := false, cnfrmExecLeft := #Axis64Pos.monitoring.interlockJogBackward, cnfrmExecRight := #Axis64Pos.monitoring.interlockJogForward, disableLeft := #disableUnit, disableRight := #disableUnit, cnfrmExecLeftCmd := #manualOperationCms.cmd.execLeftCmd, cnfrmExecRightCmd := #manualOperationCms.cmd.execRightCmd, fieldDevAckLeft := #Axis64Pos.monitoring.jogBackward, fieldDevAckRight := #Axis64Pos.monitoring.jogForward, nextLeftEndPos := 0, nextRightEndPos := 0, leftEndPosSens1 := #SoftCamInterface.posistion0.inPos, leftEndPosSens2 := #SoftCamInterface.posistion1.inPos, leftEndPosSens3 := #SoftCamInterface.posistion2.inPos, leftEndPosSens4 := #SoftCamInterface.posistion3.inPos, leftEndPosSens5 := #SoftCamInterface.posistion4.inPos, leftEndPosSens6 := #SoftCamInterface.posistion5.inPos, leftEndPosSens7 := #SoftCamInterface.posistion6.inPos, leftEndPosSens8 := #SoftCamInterface.posistion7.inPos, rightEndPosSens1 := #SoftCamInterface.posistion8.inPos, rightEndPosSens2 := #SoftCamInterface.posistion9.inPos, rightEndPosSens3 := #SoftCamInterface.posistion10.inPos, rightEndPosSens4 := #SoftCamInterface.posistion11.inPos, rightEndPosSens5 := #SoftCamInterface.posistion12.inPos, rightEndPosSens6 := #SoftCamInterface.posistion13.inPos, rightEndPosSens7 := #SoftCamInterface.posistion14.inPos, rightEndPosSens8 := #SoftCamInterface.posistion15.inPos, pos := #Axis64Pos.monitoring.actualPosition, maxPos := #tempMaxPos, minPos := 0.0, showPos := 01, line := #manualOperationCms, status => #Status, errID => #errorID)
   END_RUNG
   RUNG wire#powerrail
      I_Contact( #disableUnit )
      wire#w1
      Contact( #manualOperationCms.cmd.execRightCmd )
      Contact( #manualOperationCms.intf.cnfrmExecRightCmd )
      S_Coil( #Axis64Pos.commands.jogForward )
   END_RUNG
   RUNG wire#w1
      I_Contact( #manualOperationCms.cmd.execRightCmd )
      I_Contact( #manualOperationCms.intf.cnfrmExecRightCmd )
      R_Coil( #Axis64Pos.commands.jogForward )
   END_RUNG
   RUNG wire#w1
      Contact( #manualOperationCms.cmd.execLeftCmd )
      Contact( #manualOperationCms.intf.cnfrmExecLeftCmd )
      S_Coil( #Axis64Pos.commands.jogBackward )
   END_RUNG
   RUNG wire#w1
      I_Contact( #manualOperationCms.cmd.execLeftCmd )
      I_Contact( #manualOperationCms.intf.cnfrmExecLeftCmd )
      R_Coil( #Axis64Pos.commands.jogBackward )
   END_RUNG
   RUNG wire#powerrail
      Contact( #disableUnit )
      wire#w2
      I_Contact( #manualOperationCms.cmd.execRightCmd )
      I_Contact( #manualOperationCms.intf.cnfrmExecRightCmd )
      R_Coil( #Axis64Pos.commands.jogForward )
   END_RUNG
   RUNG wire#w2
      I_Contact( #manualOperationCms.cmd.execLeftCmd )
      I_Contact( #manualOperationCms.intf.cnfrmExecLeftCmd )
      R_Coil( #Axis64Pos.commands.jogBackward )
   END_RUNG
   // the same network as SCL:
   "LAF_ManOperationCm"(mode := 1,
                        showLine := true,
                        enableMechAddr := false,
                        expandable := true,
                        disableLineSel := false,
                        enableBigArea := false,
                        execLeftCmd := false,
                        execRightCmd := false,
                        cnfrmExecLeft := #Axis64Pos.monitoring.interlockJogBackward,
                        cnfrmExecRight := #Axis64Pos.monitoring.interlockJogForward,
                        disableLeft := #disableUnit,
                        disableRight := #disableUnit,
                        cnfrmExecLeftCmd := #manualOperationCms.cmd.execLeftCmd,
                        cnfrmExecRightCmd := #manualOperationCms.cmd.execRightCmd,
                        fieldDevAckLeft := #Axis64Pos.monitoring.jogBackward,
                        fieldDevAckRight := #Axis64Pos.monitoring.jogForward,
                        nextLeftEndPos := 0,
                        nextRightEndPos := 0,
                        leftEndPosSens1 := #SoftCamInterface.posistion0.inPos,
                        leftEndPosSens2 := #SoftCamInterface.posistion1.inPos,
                        leftEndPosSens3 := #SoftCamInterface.posistion2.inPos,
                        leftEndPosSens4 := #SoftCamInterface.posistion3.inPos,
                        leftEndPosSens5 := #SoftCamInterface.posistion4.inPos,
                        leftEndPosSens6 := #SoftCamInterface.posistion5.inPos,
                        leftEndPosSens7 := #SoftCamInterface.posistion6.inPos,
                        leftEndPosSens8 := #SoftCamInterface.posistion7.inPos,
                        rightEndPosSens1 := #SoftCamInterface.posistion8.inPos,
                        rightEndPosSens2 := #SoftCamInterface.posistion9.inPos,
                        rightEndPosSens3 := #SoftCamInterface.posistion10.inPos,
                        rightEndPosSens4 := #SoftCamInterface.posistion11.inPos,
                        rightEndPosSens5 := #SoftCamInterface.posistion12.inPos,
                        rightEndPosSens6 := #SoftCamInterface.posistion13.inPos,
                        rightEndPosSens7 := #SoftCamInterface.posistion14.inPos,
                        rightEndPosSens8 := #SoftCamInterface.posistion15.inPos,
                        pos := #Axis64Pos.monitoring.actualPosition,
                        maxPos := #tempMaxPos,
                        minPos := 0.0,
                        showPos := 01,
                        line := #manualOperationCms,
                        status => #Status,
                        errID => #errorID);
   IF NOT #disableUnit AND #manualOperationCms.cmd.execRightCmd AND #manualOperationCms.intf.cnfrmExecRightCmd THEN
       #Axis64Pos.commands.jogForward := TRUE;
   END_IF;
   IF NOT #disableUnit AND NOT #manualOperationCms.cmd.execRightCmd AND NOT #manualOperationCms.intf.cnfrmExecRightCmd THEN
       #Axis64Pos.commands.jogForward := FALSE;
   END_IF;
   IF NOT #disableUnit AND #manualOperationCms.cmd.execLeftCmd AND #manualOperationCms.intf.cnfrmExecLeftCmd THEN
       #Axis64Pos.commands.jogBackward := TRUE;
   END_IF;
   IF NOT #disableUnit AND NOT #manualOperationCms.cmd.execLeftCmd AND NOT #manualOperationCms.intf.cnfrmExecLeftCmd THEN
       #Axis64Pos.commands.jogBackward := FALSE;
   END_IF;
   IF #disableUnit AND NOT #manualOperationCms.cmd.execRightCmd AND NOT #manualOperationCms.intf.cnfrmExecRightCmd THEN
       #Axis64Pos.commands.jogForward := FALSE;
   END_IF;
   IF #disableUnit AND NOT #manualOperationCms.cmd.execLeftCmd AND NOT #manualOperationCms.intf.cnfrmExecLeftCmd THEN
       #Axis64Pos.commands.jogBackward := FALSE;
   END_IF;
END_REGION
END_FUNCTION

FUNCTION "ManOperationCm_typeTwoWayActuatorInterface" : Void   // FC65, LAD
// stored: SetENOAutomatically false
   VAR_INPUT
      disableUnit : Bool;
   END_VAR
   VAR_OUTPUT
      Status : Word;
      errorID : Word;
   END_VAR
   VAR_IN_OUT
      manualOperationEm : "LAF_typeManEm";
      manualOperationEmArea : "LAF_typeManOperationArea";
      manualOperationCms : "LAF_typeManOperation";
      twoWayAcutor : "LBC_typeTwoWayActuatorInterface";
   END_VAR
BEGIN

REGION Network 1: Manual Operation Cm - typeTwoWayActuatorInterface
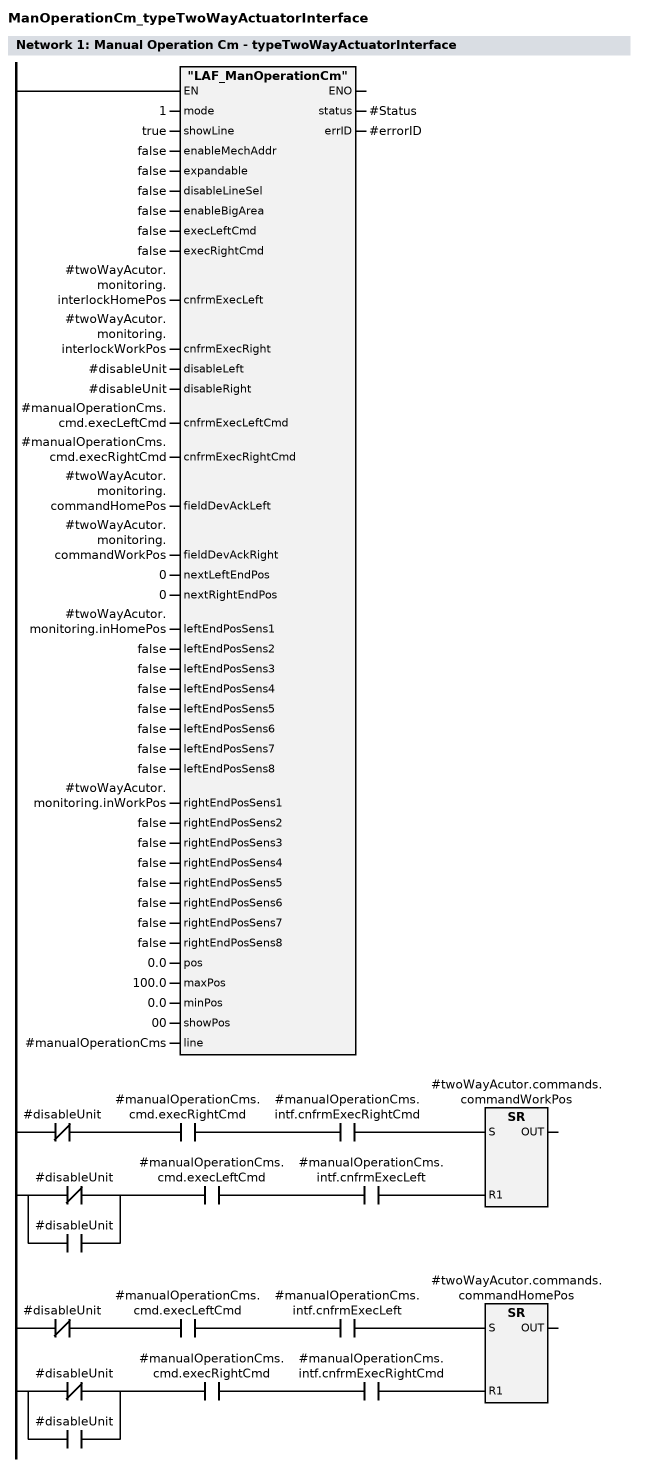
   RUNG wire#powerrail
      "LAF_ManOperationCm"(mode := 1, showLine := true, enableMechAddr := false, expandable := false, disableLineSel := false, enableBigArea := false, execLeftCmd := false, execRightCmd := false, cnfrmExecLeft := #twoWayAcutor.monitoring.interlockHomePos, cnfrmExecRight := #twoWayAcutor.monitoring.interlockWorkPos, disableLeft := #disableUnit, disableRight := #disableUnit, cnfrmExecLeftCmd := #manualOperationCms.cmd.execLeftCmd, cnfrmExecRightCmd := #manualOperationCms.cmd.execRightCmd, fieldDevAckLeft := #twoWayAcutor.monitoring.commandHomePos, fieldDevAckRight := #twoWayAcutor.monitoring.commandWorkPos, nextLeftEndPos := 0, nextRightEndPos := 0, leftEndPosSens1 := #twoWayAcutor.monitoring.inHomePos, leftEndPosSens2 := false, leftEndPosSens3 := false, leftEndPosSens4 := false, leftEndPosSens5 := false, leftEndPosSens6 := false, leftEndPosSens7 := false, leftEndPosSens8 := false, rightEndPosSens1 := #twoWayAcutor.monitoring.inWorkPos, rightEndPosSens2 := false, rightEndPosSens3 := false, rightEndPosSens4 := false, rightEndPosSens5 := false, rightEndPosSens6 := false, rightEndPosSens7 := false, rightEndPosSens8 := false, pos := 0.0, maxPos := 100.0, minPos := 0.0, showPos := 00, line := #manualOperationCms, status => #Status, errID => #errorID)
   END_RUNG
   RUNG wire#powerrail
      I_Contact( #disableUnit )
      Contact( #manualOperationCms.cmd.execRightCmd )
      Contact( #manualOperationCms.intf.cnfrmExecRightCmd )
      S_SR(operand := #twoWayAcutor.commands.commandWorkPos, r1 := wire#w2)
   END_RUNG
   RUNG wire#powerrail
      I_Contact( #disableUnit )
      wire#w1
      Contact( #manualOperationCms.cmd.execLeftCmd )
      Contact( #manualOperationCms.intf.cnfrmExecLeft )
   END_RUNG wire#w2
   RUNG wire#powerrail
      Contact( #disableUnit )
   END_RUNG wire#w1
   RUNG wire#powerrail
      I_Contact( #disableUnit )
      Contact( #manualOperationCms.cmd.execLeftCmd )
      Contact( #manualOperationCms.intf.cnfrmExecLeft )
      S_SR(operand := #twoWayAcutor.commands.commandHomePos, r1 := wire#w4)
   END_RUNG
   RUNG wire#powerrail
      I_Contact( #disableUnit )
      wire#w3
      Contact( #manualOperationCms.cmd.execRightCmd )
      Contact( #manualOperationCms.intf.cnfrmExecRightCmd )
   END_RUNG wire#w4
   RUNG wire#powerrail
      Contact( #disableUnit )
   END_RUNG wire#w3
   // the same network as SCL:
   "LAF_ManOperationCm"(mode := 1,
                        showLine := true,
                        enableMechAddr := false,
                        expandable := false,
                        disableLineSel := false,
                        enableBigArea := false,
                        execLeftCmd := false,
                        execRightCmd := false,
                        cnfrmExecLeft := #twoWayAcutor.monitoring.interlockHomePos,
                        cnfrmExecRight := #twoWayAcutor.monitoring.interlockWorkPos,
                        disableLeft := #disableUnit,
                        disableRight := #disableUnit,
                        cnfrmExecLeftCmd := #manualOperationCms.cmd.execLeftCmd,
                        cnfrmExecRightCmd := #manualOperationCms.cmd.execRightCmd,
                        fieldDevAckLeft := #twoWayAcutor.monitoring.commandHomePos,
                        fieldDevAckRight := #twoWayAcutor.monitoring.commandWorkPos,
                        nextLeftEndPos := 0,
                        nextRightEndPos := 0,
                        leftEndPosSens1 := #twoWayAcutor.monitoring.inHomePos,
                        leftEndPosSens2 := false,
                        leftEndPosSens3 := false,
                        leftEndPosSens4 := false,
                        leftEndPosSens5 := false,
                        leftEndPosSens6 := false,
                        leftEndPosSens7 := false,
                        leftEndPosSens8 := false,
                        rightEndPosSens1 := #twoWayAcutor.monitoring.inWorkPos,
                        rightEndPosSens2 := false,
                        rightEndPosSens3 := false,
                        rightEndPosSens4 := false,
                        rightEndPosSens5 := false,
                        rightEndPosSens6 := false,
                        rightEndPosSens7 := false,
                        rightEndPosSens8 := false,
                        pos := 0.0,
                        maxPos := 100.0,
                        minPos := 0.0,
                        showPos := 00,
                        line := #manualOperationCms,
                        status => #Status,
                        errID => #errorID);
   IF NOT #disableUnit AND #manualOperationCms.cmd.execRightCmd AND #manualOperationCms.intf.cnfrmExecRightCmd THEN
       #twoWayAcutor.commands.commandWorkPos := TRUE;   // SR flip-flop
   END_IF;
   IF (NOT #disableUnit OR #disableUnit) AND #manualOperationCms.cmd.execLeftCmd AND #manualOperationCms.intf.cnfrmExecLeft THEN
       #twoWayAcutor.commands.commandWorkPos := FALSE;
   END_IF;
   IF NOT #disableUnit AND #manualOperationCms.cmd.execLeftCmd AND #manualOperationCms.intf.cnfrmExecLeft THEN
       #twoWayAcutor.commands.commandHomePos := TRUE;   // SR flip-flop
   END_IF;
   IF (NOT #disableUnit OR #disableUnit) AND #manualOperationCms.cmd.execRightCmd AND #manualOperationCms.intf.cnfrmExecRightCmd THEN
       #twoWayAcutor.commands.commandHomePos := FALSE;
   END_IF;
END_REGION
END_FUNCTION

FUNCTION "CallDiagnostic" : Void   // FC16, LAD
TITLE = Diagnose / Diagnostics
AUTHOR : SICAR
FAMILY : Diag
// Aufruf: Diagnose / Call of SICAR Diagnostic blocks
// stored: IsIECCheckEnabled true, SetENOAutomatically true
   VAR_TEMP
      statWStringName : WString[24];
      tempHardwareOKexample : Bool;   // REPLACE: This output can be used as an interlock for Control Modules
   END_VAR
   // Ret_Val : Ret_Val
   VAR_TEMP   // added for the SCL form of the ladder/FBD networks
      _w1 : Bool;
   END_VAR
BEGIN

REGION Network 1: Beschreibung / BLOCK INFO HEADER
   // **Betriebsart Automatik / Hand**  
   // Der Baustein ist keiner Betriebsart / Betriebsartenbereich zugeordnet.  
   // 
   // **Alarme**  
   // Der Baustein generiert keine Alarme.  
   // 
   // #### PLC-Datentypen  
   // Verwendete PLC-Datentypen für den SPS-Programmbaustein und das zugehörige WinCC-Bild.  
   // 
   // {.pageWidth}
   // ![Image](CallInterfaceSignals/de/image1.PNG)
   //  
   //  
   // #### Bausteinaufrufe 
   // Der Baustein “LSicar_InterfaceSignalsBool“ wird in diesem FB als Multi-Instanz aufgerufen, entspr. nebenstehender beispielhafter Darstellung.  
   // 
   // {.pageWidth}
   // ![Image](CallInterfaceSignals/de/image2.PNG)
   //  
   // Um einen neuen FB aufzurufen, ziehen Sie den FB in ein neues Netzwerk, wählen Sie „Multiinstanz“ aus, vergeben Sie einen Namen und parametrieren Sie den FB-Aufruf.  
   // 
   // {.pageWidth}
   // ![Image](CallInterfaceSignals/de/image3.PNG)
   //  
   //  
   // #### Weitere Hinweise 
   // 
   // #### Updateinfo 
   // 
   // #### Weitere Dokumente 
   // 
   // ![Icon](_Icon/reference.PNG)
   // 
   // ..\Library Types\LSicar_InterfaceSignalsBool.pdf
   // SIEMENS AG / (c)Copyright 2023
   // ------------------------------------------------------------------------------
   // Title:            CallDiagnostic (FC16)
   // Comment/Function: Call of SICAR Diagnostic blocks
   // Library/Family:   Diag
   // Author:           SICAR
   // Tested with:      ---
   // Engineering:      TIA Portal V19
   // Restrictions:     -
   // Requirements:     ---
   // ------------------------------------------------------------------------------
   // Change log table:
   // Version | Date | Expert in charge | Changes applied
   // -------|---------|-------------|--------------------------------------------
   // 01.00.00 | 01.01.1999 | Person x | First released version
   // 01.00.01 | 02.01.1999 | Person y | Block was Updated
END_REGION

